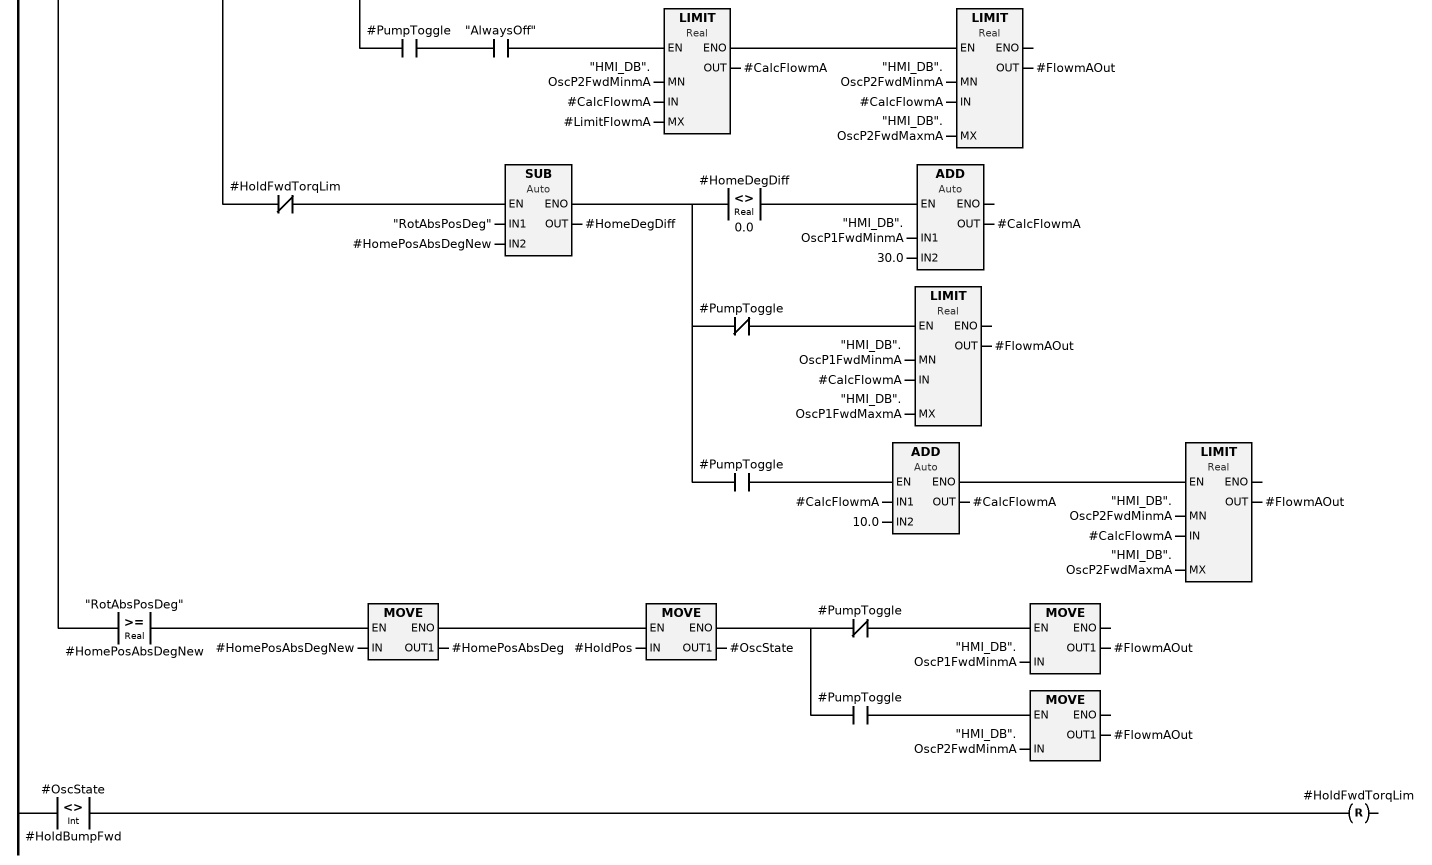
   RUNG wire#powerrail
      { S7_Templates := "SrcType := Int" } EQ_Contact(in1 := #OscState, in2 := #HoldBumpFwd)
      wire#w1
      Contact( #Oscillating )
      wire#w2
      P_Trig( #BumpFwdTrig )
      Move(in := "RotAbsPosDeg", out1 => #StartDeg)
      wire#w3
      I_Contact( #PumpToggle )
      Move(in := "HMI_DB".OscP1FwdMinmA, out1 => #CalcFlowmA)
   END_RUNG
   RUNG wire#w1
      Contact( #Holding )
   END_RUNG wire#w2
   RUNG wire#w3
      Contact( #PumpToggle )
      Move(in := "HMI_DB".OscP2FwdMinmA, out1 => #CalcFlowmA)
   END_RUNG
   RUNG wire#w2
      R_Coil( #FlowRev )
   END_RUNG
   RUNG wire#w2
      R_Coil( "HMI_DB".OscBumpFwd )
   END_RUNG
   RUNG wire#w2
      { S7_Templates := "SrcType := Real" } LT_Contact(in1 := "RotAbsPosDeg", in2 := #HomePosAbsDegNew)
      wire#w4
      { S7_Templates := "SrcType := Real" } GE_Contact(in1 := "ActTorqFtLbsFilt", in2 := "HMI_DB".OscTorqFwdLowLimFtlbs)
      { S7_Templates := "time_type := Time" } #HoldFWDTorqLim_TON.TON(pt := "Settings".OscTorqLimTime, et =>)
      S_Coil( #HoldFwdTorqLim )
   END_RUNG
   RUNG wire#w4
      { S7_Templates := "SrcType := Real" } GE_Contact(in1 := "ActTorqFtLbsFilt", in2 := "HMI_DB".OscTorqFwdHighLimFtLbs)
      S_Coil( #HoldFwdTorqLim )
   END_RUNG
   RUNG wire#w4
      Contact( #HoldFwdTorqLim )
      P_Trig( #HoldFwdTorqLimTrig )
      Move(in := #CalcFlowmA, out1 => #LimitFlowmA)
   END_RUNG
   RUNG wire#w4
      { S7_Templates := "SrcType := Real" } LT_Contact(in1 := "ActTorqFtLbsFilt", in2 := "HMI_DB".OscTorqFwdLowLimFtlbs)
      { S7_Templates := "SrcType := Real" } LT_Contact(in1 := #CalcFlowmA, in2 := #LimitFlowmA)
      R_Coil( #HoldFwdTorqLim )
   END_RUNG
   RUNG wire#w4
      Contact( #HoldFwdTorqLim )
      wire#w5
      { S7_Templates := "SrcType := Real" } GE_Contact(in1 := "ActTorqFtLbsFilt", in2 := "HMI_DB".OscTorqFwdHighLimFtLbs)
      Contact( "AlwaysOff" )
      #HoldFwdTorqLim_SlewDec(SlewRate := "HMI_DB".OscSlewFallSlow, RealValue := #LimitFlowmA)
   END_RUNG
   RUNG wire#w5
      { S7_Templates := "SrcType := Real" } LT_Contact(in1 := "ActTorqFtLbsFilt", in2 := "HMI_DB".OscTorqFwdLowLimFtlbs)
      Contact( "AlwaysOff" )
      #HoldFwdTorqLim_SlewInc(SlewRate := "HMI_DB".OscSlewRiseSlow, RealValue := #LimitFlowmA)
   END_RUNG
   RUNG wire#w5
      I_Contact( #PumpToggle )
      Contact( "AlwaysOff" )
      { S7_Templates := "value_type := Real" } Limit(mn := "HMI_DB".OscP1FwdMinmA, in := #CalcFlowmA, mx := #LimitFlowmA, out => #CalcFlowmA)
      { S7_Templates := "value_type := Real" } Limit(mn := "HMI_DB".OscP1FwdMinmA, in := #CalcFlowmA, mx := "HMI_DB".OscP1FwdMaxmA, out => #FlowmAOut)
   END_RUNG
   RUNG wire#w5
      Contact( #PumpToggle )
      Contact( "AlwaysOff" )
      { S7_Templates := "value_type := Real" } Limit(mn := "HMI_DB".OscP2FwdMinmA, in := #CalcFlowmA, mx := #LimitFlowmA, out => #CalcFlowmA)
      { S7_Templates := "value_type := Real" } Limit(mn := "HMI_DB".OscP2FwdMinmA, in := #CalcFlowmA, mx := "HMI_DB".OscP2FwdMaxmA, out => #FlowmAOut)
   END_RUNG
   RUNG wire#w4
      I_Contact( #HoldFwdTorqLim )
      Sub(in1 := "RotAbsPosDeg", in2 := #HomePosAbsDegNew, out => #HomeDegDiff)
      wire#w6
      { S7_Templates := "SrcType := Real" } NE_Contact(in1 := #HomeDegDiff, in2 := 0.0)
      Add(in1 := "HMI_DB".OscP1FwdMinmA, in2 := 30.0, out => #CalcFlowmA)
   END_RUNG
   RUNG wire#w6
      I_Contact( #PumpToggle )
      { S7_Templates := "value_type := Real" } Limit(mn := "HMI_DB".OscP1FwdMinmA, in := #CalcFlowmA, mx := "HMI_DB".OscP1FwdMaxmA, out => #FlowmAOut)
   END_RUNG
   RUNG wire#w6
      Contact( #PumpToggle )
      Add(in1 := #CalcFlowmA, in2 := 10.0, out => #CalcFlowmA)
      { S7_Templates := "value_type := Real" } Limit(mn := "HMI_DB".OscP2FwdMinmA, in := #CalcFlowmA, mx := "HMI_DB".OscP2FwdMaxmA, out => #FlowmAOut)
   END_RUNG
   RUNG wire#w2
      { S7_Templates := "SrcType := Real" } GE_Contact(in1 := "RotAbsPosDeg", in2 := #HomePosAbsDegNew)
      Move(in := #HomePosAbsDegNew, out1 => #HomePosAbsDeg)
      Move(in := #HoldPos, out1 => #OscState)
      wire#w7
      I_Contact( #PumpToggle )
      Move(in := "HMI_DB".OscP1FwdMinmA, out1 => #FlowmAOut)
   END_RUNG
   RUNG wire#w7
      Contact( #PumpToggle )
      Move(in := "HMI_DB".OscP2FwdMinmA, out1 => #FlowmAOut)
   END_RUNG
   RUNG wire#powerrail
      { S7_Templates := "SrcType := Int" } NE_Contact(in1 := #OscState, in2 := #HoldBumpFwd)
      R_Coil( #HoldFwdTorqLim )
   END_RUNG
   // the same network as SCL:
   #_w1 := (#OscState = #HoldBumpFwd) AND (#Oscillating OR #Holding);
   #_w2 := #_w1 AND NOT #BumpFwdTrig;   // rising edge
   #BumpFwdTrig := #_w1;
   IF #_w2 THEN #StartDeg := "RotAbsPosDeg"; END_IF;
   IF #_w2 AND NOT #PumpToggle THEN #CalcFlowmA := "HMI_DB".OscP1FwdMinmA; END_IF;
   IF #_w2 AND #PumpToggle THEN #CalcFlowmA := "HMI_DB".OscP2FwdMinmA; END_IF;
   IF #_w1 THEN
       #FlowRev := FALSE;
       "HMI_DB".OscBumpFwd := FALSE;
   END_IF;
   #_w3 := #_w1 AND ("RotAbsPosDeg" < #HomePosAbsDegNew);
   #HoldFWDTorqLim_TON(IN := #_w3 AND ("ActTorqFtLbsFilt" >= "HMI_DB".OscTorqFwdLowLimFtlbs),   // TON
                       PT := "Settings".OscTorqLimTime);
   IF #HoldFWDTorqLim_TON.Q THEN #HoldFwdTorqLim := TRUE; END_IF;
   IF #_w3 AND ("ActTorqFtLbsFilt" >= "HMI_DB".OscTorqFwdHighLimFtLbs) THEN #HoldFwdTorqLim := TRUE; END_IF;
   #_w4 := #_w3 AND #HoldFwdTorqLim;
   #_w5 := #_w4 AND NOT #HoldFwdTorqLimTrig;   // rising edge
   #HoldFwdTorqLimTrig := #_w4;
   IF #_w5 THEN #LimitFlowmA := #CalcFlowmA; END_IF;
   IF #_w3 AND ("ActTorqFtLbsFilt" < "HMI_DB".OscTorqFwdLowLimFtlbs) AND (#CalcFlowmA < #LimitFlowmA) THEN
       #HoldFwdTorqLim := FALSE;
   END_IF;
   #_w6 := #_w3 AND #HoldFwdTorqLim;
   IF #_w6 AND ("ActTorqFtLbsFilt" >= "HMI_DB".OscTorqFwdHighLimFtLbs) AND "AlwaysOff" THEN
       #HoldFwdTorqLim_SlewDec(SlewRate := "HMI_DB".OscSlewFallSlow, RealValue := #LimitFlowmA);   // "SlewDec"
   END_IF;
   IF #_w6 AND ("ActTorqFtLbsFilt" < "HMI_DB".OscTorqFwdLowLimFtlbs) AND "AlwaysOff" THEN
       #HoldFwdTorqLim_SlewInc(SlewRate := "HMI_DB".OscSlewRiseSlow, RealValue := #LimitFlowmA);   // "SlewInc"
   END_IF;
   IF #_w6 AND NOT #PumpToggle AND "AlwaysOff" THEN
       #CalcFlowmA := LIMIT(MN := "HMI_DB".OscP1FwdMinmA, IN := #CalcFlowmA, MX := #LimitFlowmA);
       #FlowmAOut := LIMIT(MN := "HMI_DB".OscP1FwdMinmA, IN := #CalcFlowmA, MX := "HMI_DB".OscP1FwdMaxmA);
   END_IF;
   IF #_w6 AND #PumpToggle AND "AlwaysOff" THEN
       #CalcFlowmA := LIMIT(MN := "HMI_DB".OscP2FwdMinmA, IN := #CalcFlowmA, MX := #LimitFlowmA);
       #FlowmAOut := LIMIT(MN := "HMI_DB".OscP2FwdMinmA, IN := #CalcFlowmA, MX := "HMI_DB".OscP2FwdMaxmA);
   END_IF;
   #_w7 := #_w3 AND NOT #HoldFwdTorqLim;
   IF #_w7 THEN #HomeDegDiff := "RotAbsPosDeg" - #HomePosAbsDegNew; END_IF;
   IF #_w7 AND (#HomeDegDiff <> 0.0) THEN #CalcFlowmA := "HMI_DB".OscP1FwdMinmA + 30.0; END_IF;
   IF #_w7 AND NOT #PumpToggle THEN
       #FlowmAOut := LIMIT(MN := "HMI_DB".OscP1FwdMinmA, IN := #CalcFlowmA, MX := "HMI_DB".OscP1FwdMaxmA);
   END_IF;
   IF #_w7 AND #PumpToggle THEN
       #CalcFlowmA := #CalcFlowmA + 10.0;
       #FlowmAOut := LIMIT(MN := "HMI_DB".OscP2FwdMinmA, IN := #CalcFlowmA, MX := "HMI_DB".OscP2FwdMaxmA);
   END_IF;
   #_w8 := #_w1 AND ("RotAbsPosDeg" >= #HomePosAbsDegNew);
   IF #_w8 THEN
       #HomePosAbsDeg := #HomePosAbsDegNew;
       #OscState := #HoldPos;
   END_IF;
   IF #_w8 AND NOT #PumpToggle THEN #FlowmAOut := "HMI_DB".OscP1FwdMinmA; END_IF;
   IF #_w8 AND #PumpToggle THEN #FlowmAOut := "HMI_DB".OscP2FwdMinmA; END_IF;
   IF #OscState <> #HoldBumpFwd THEN #HoldFwdTorqLim := FALSE; END_IF;
END_REGION

REGION Network 11: Hold Bump Reactive - State 104
   // Allow the quill to reactively move to the new position. 
   // Flow Rev enabled to Min until at Home position. If position below start position, min too high and moving wrong direction. Not reacting.  
   // At or above new home position, hold position
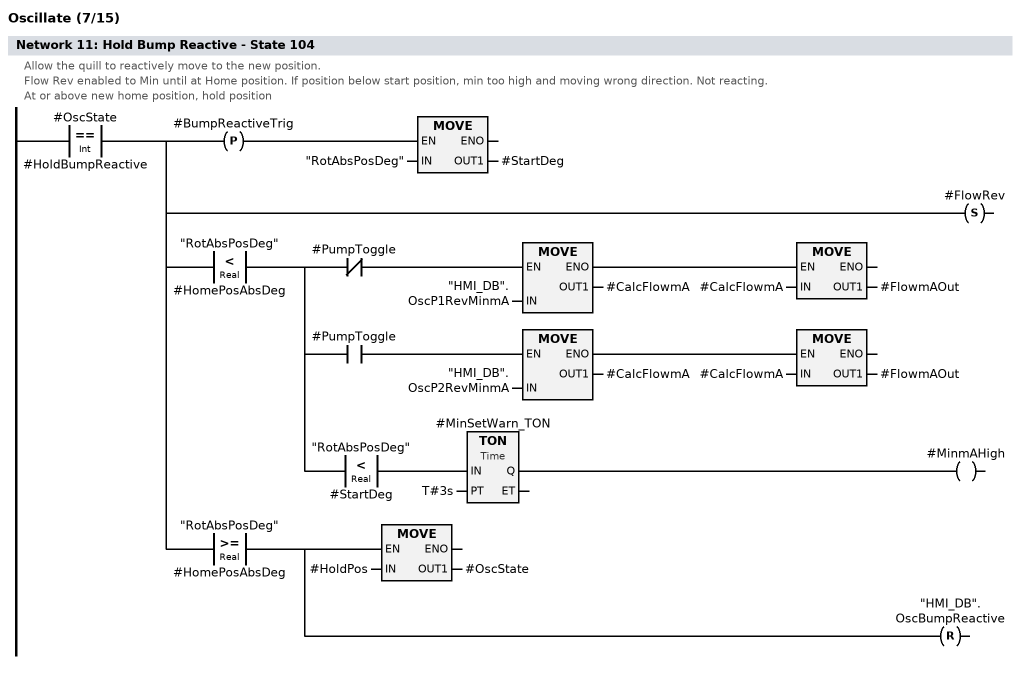
   RUNG wire#powerrail
      { S7_Templates := "SrcType := Int" } EQ_Contact(in1 := #OscState, in2 := #HoldBumpReactive)
      wire#w1
      P_Trig( #BumpReactiveTrig )
      Move(in := "RotAbsPosDeg", out1 => #StartDeg)
   END_RUNG
   RUNG wire#w1
      S_Coil( #FlowRev )
   END_RUNG
   RUNG wire#w1
      { S7_Templates := "SrcType := Real" } LT_Contact(in1 := "RotAbsPosDeg", in2 := #HomePosAbsDeg)
      wire#w2
      I_Contact( #PumpToggle )
      Move(in := "HMI_DB".OscP1RevMinmA, out1 => #CalcFlowmA)
      Move(in := #CalcFlowmA, out1 => #FlowmAOut)
   END_RUNG
   RUNG wire#w2
      Contact( #PumpToggle )
      Move(in := "HMI_DB".OscP2RevMinmA, out1 => #CalcFlowmA)
      Move(in := #CalcFlowmA, out1 => #FlowmAOut)
   END_RUNG
   RUNG wire#w2
      { S7_Templates := "SrcType := Real" } LT_Contact(in1 := "RotAbsPosDeg", in2 := #StartDeg)
      { S7_Templates := "time_type := Time" } #MinSetWarn_TON.TON(pt := T#3s, et =>)
      Coil( #MinmAHigh )
   END_RUNG
   RUNG wire#w1
      { S7_Templates := "SrcType := Real" } GE_Contact(in1 := "RotAbsPosDeg", in2 := #HomePosAbsDeg)
      wire#w3
      Move(in := #HoldPos, out1 => #OscState)
   END_RUNG
   RUNG wire#w3
      R_Coil( "HMI_DB".OscBumpReactive )
   END_RUNG
   // the same network as SCL:
   #_w1 := #OscState = #HoldBumpReactive;
   #_w2 := #_w1 AND NOT #BumpReactiveTrig;   // rising edge
   #BumpReactiveTrig := #_w1;
   IF #_w2 THEN #StartDeg := "RotAbsPosDeg"; END_IF;
   IF #_w1 THEN #FlowRev := TRUE; END_IF;
   #_w3 := #_w1 AND ("RotAbsPosDeg" < #HomePosAbsDeg);
   IF #_w3 AND NOT #PumpToggle THEN
       #CalcFlowmA := "HMI_DB".OscP1RevMinmA;
       #FlowmAOut := #CalcFlowmA;
   END_IF;
   IF #_w3 AND #PumpToggle THEN
       #CalcFlowmA := "HMI_DB".OscP2RevMinmA;
       #FlowmAOut := #CalcFlowmA;
   END_IF;
   #MinSetWarn_TON(IN := #_w3 AND ("RotAbsPosDeg" < #StartDeg), PT := T#3s);   // TON
   #MinmAHigh := #MinSetWarn_TON.Q;
   IF #_w1 AND ("RotAbsPosDeg" >= #HomePosAbsDeg) THEN
       #OscState := #HoldPos;
       "HMI_DB".OscBumpReactive := FALSE;
   END_IF;
END_REGION

REGION Network 12: Hold Bump Rev - State 103
   // Move quill to new position in the Rev direction. 
   // Start at Hold mA and Ramp up until speed reach. 
   // If Approaching Torq Limit, limit output flow. 
   // At or above new home position, output hold value and hold position
   // Note: Dummy Move On Maintain speed there as visual only.
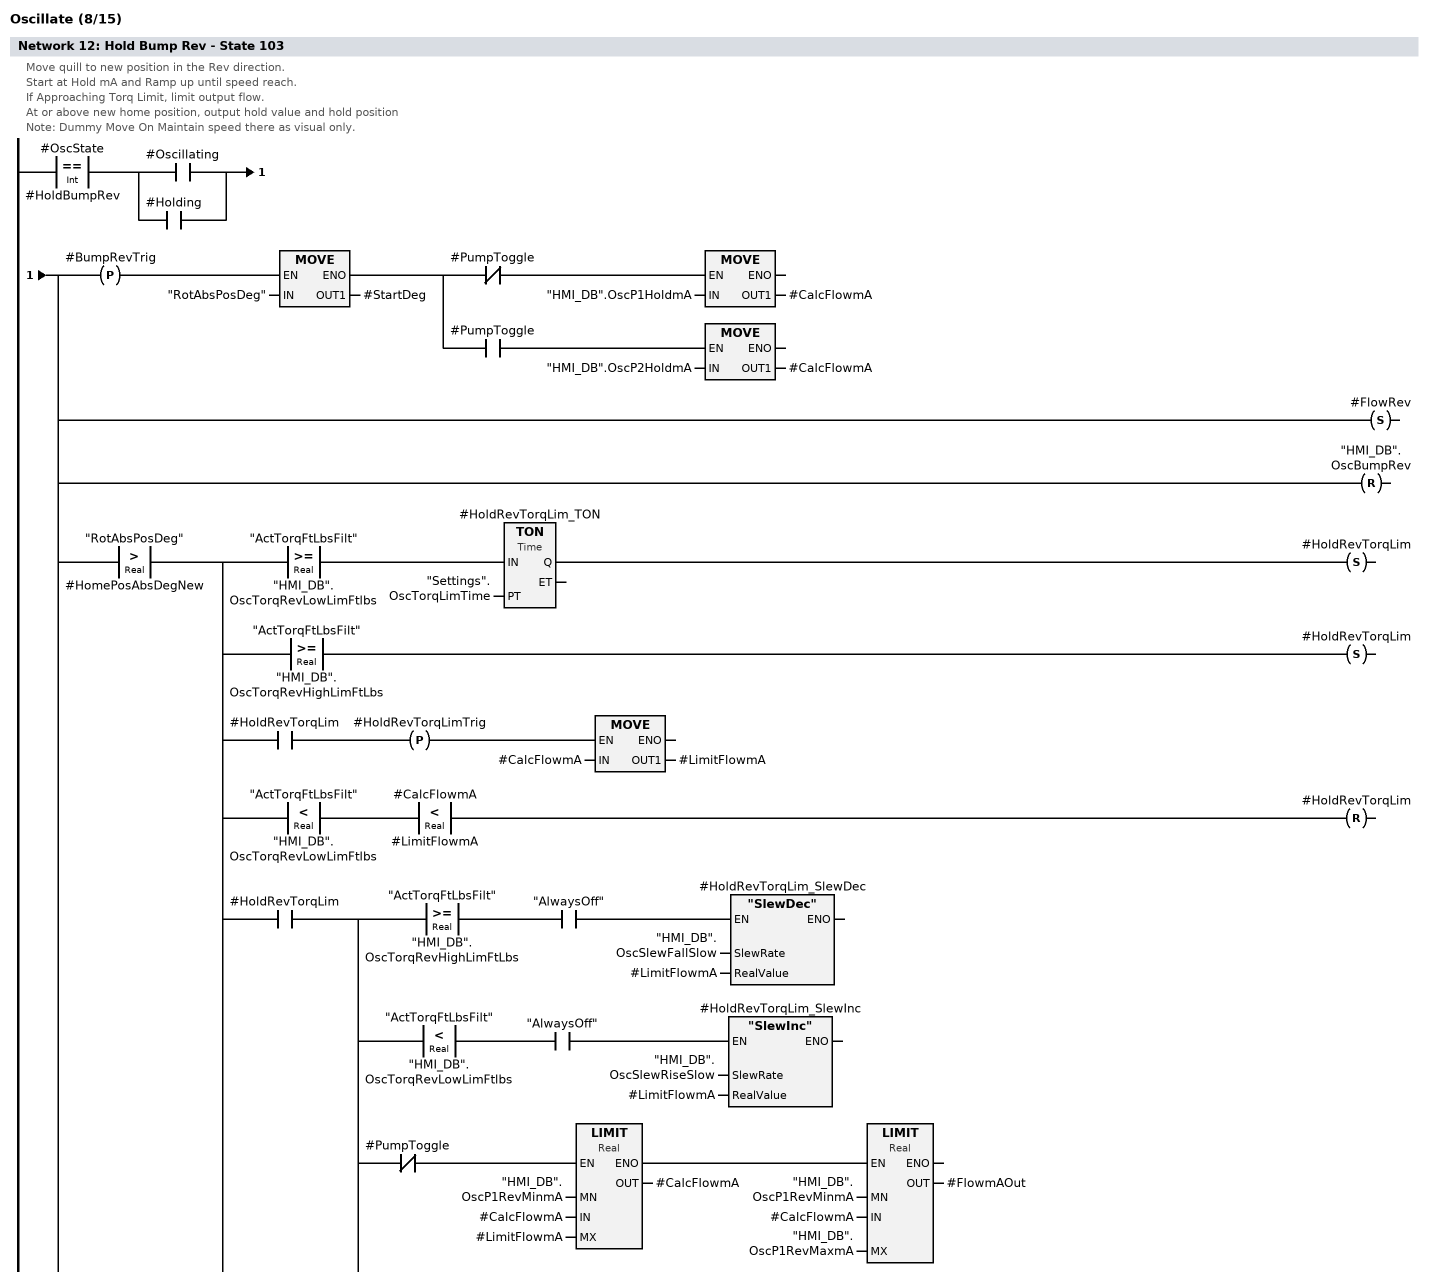
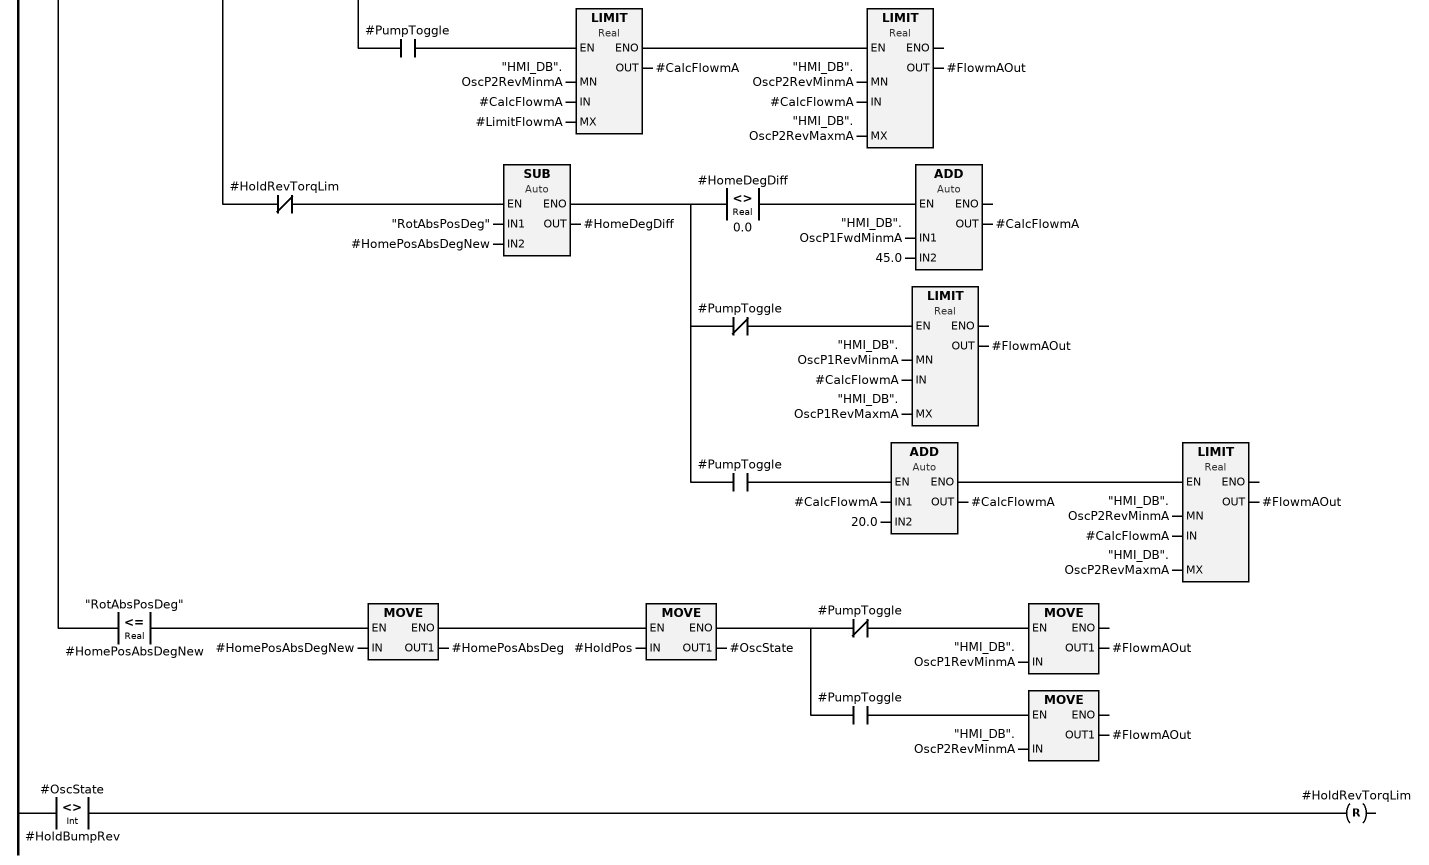
   RUNG wire#powerrail
      { S7_Templates := "SrcType := Int" } EQ_Contact(in1 := #OscState, in2 := #HoldBumpRev)
      wire#w1
      Contact( #Oscillating )
      wire#w2
      P_Trig( #BumpRevTrig )
      Move(in := "RotAbsPosDeg", out1 => #StartDeg)
      wire#w3
      I_Contact( #PumpToggle )
      Move(in := "HMI_DB".OscP1HoldmA, out1 => #CalcFlowmA)
   END_RUNG
   RUNG wire#w1
      Contact( #Holding )
   END_RUNG wire#w2
   RUNG wire#w3
      Contact( #PumpToggle )
      Move(in := "HMI_DB".OscP2HoldmA, out1 => #CalcFlowmA)
   END_RUNG
   RUNG wire#w2
      S_Coil( #FlowRev )
   END_RUNG
   RUNG wire#w2
      R_Coil( "HMI_DB".OscBumpRev )
   END_RUNG
   RUNG wire#w2
      { S7_Templates := "SrcType := Real" } GT_Contact(in1 := "RotAbsPosDeg", in2 := #HomePosAbsDegNew)
      wire#w4
      { S7_Templates := "SrcType := Real" } GE_Contact(in1 := "ActTorqFtLbsFilt", in2 := "HMI_DB".OscTorqRevLowLimFtlbs)
      { S7_Templates := "time_type := Time" } #HoldRevTorqLim_TON.TON(pt := "Settings".OscTorqLimTime, et =>)
      S_Coil( #HoldRevTorqLim )
   END_RUNG
   RUNG wire#w4
      { S7_Templates := "SrcType := Real" } GE_Contact(in1 := "ActTorqFtLbsFilt", in2 := "HMI_DB".OscTorqRevHighLimFtLbs)
      S_Coil( #HoldRevTorqLim )
   END_RUNG
   RUNG wire#w4
      Contact( #HoldRevTorqLim )
      P_Trig( #HoldRevTorqLimTrig )
      Move(in := #CalcFlowmA, out1 => #LimitFlowmA)
   END_RUNG
   RUNG wire#w4
      { S7_Templates := "SrcType := Real" } LT_Contact(in1 := "ActTorqFtLbsFilt", in2 := "HMI_DB".OscTorqRevLowLimFtlbs)
      { S7_Templates := "SrcType := Real" } LT_Contact(in1 := #CalcFlowmA, in2 := #LimitFlowmA)
      R_Coil( #HoldRevTorqLim )
   END_RUNG
   RUNG wire#w4
      Contact( #HoldRevTorqLim )
      wire#w5
      { S7_Templates := "SrcType := Real" } GE_Contact(in1 := "ActTorqFtLbsFilt", in2 := "HMI_DB".OscTorqRevHighLimFtLbs)
      Contact( "AlwaysOff" )
      #HoldRevTorqLim_SlewDec(SlewRate := "HMI_DB".OscSlewFallSlow, RealValue := #LimitFlowmA)
   END_RUNG
   RUNG wire#w5
      { S7_Templates := "SrcType := Real" } LT_Contact(in1 := "ActTorqFtLbsFilt", in2 := "HMI_DB".OscTorqRevLowLimFtlbs)
      Contact( "AlwaysOff" )
      #HoldRevTorqLim_SlewInc(SlewRate := "HMI_DB".OscSlewRiseSlow, RealValue := #LimitFlowmA)
   END_RUNG
   RUNG wire#w5
      I_Contact( #PumpToggle )
      { S7_Templates := "value_type := Real" } Limit(mn := "HMI_DB".OscP1RevMinmA, in := #CalcFlowmA, mx := #LimitFlowmA, out => #CalcFlowmA)
      { S7_Templates := "value_type := Real" } Limit(mn := "HMI_DB".OscP1RevMinmA, in := #CalcFlowmA, mx := "HMI_DB".OscP1RevMaxmA, out => #FlowmAOut)
   END_RUNG
   RUNG wire#w5
      Contact( #PumpToggle )
      { S7_Templates := "value_type := Real" } Limit(mn := "HMI_DB".OscP2RevMinmA, in := #CalcFlowmA, mx := #LimitFlowmA, out => #CalcFlowmA)
      { S7_Templates := "value_type := Real" } Limit(mn := "HMI_DB".OscP2RevMinmA, in := #CalcFlowmA, mx := "HMI_DB".OscP2RevMaxmA, out => #FlowmAOut)
   END_RUNG
   RUNG wire#w4
      I_Contact( #HoldRevTorqLim )
      Sub(in1 := "RotAbsPosDeg", in2 := #HomePosAbsDegNew, out => #HomeDegDiff)
      wire#w6
      { S7_Templates := "SrcType := Real" } NE_Contact(in1 := #HomeDegDiff, in2 := 0.0)
      Add(in1 := "HMI_DB".OscP1FwdMinmA, in2 := 45.0, out => #CalcFlowmA)
   END_RUNG
   RUNG wire#w6
      I_Contact( #PumpToggle )
      { S7_Templates := "value_type := Real" } Limit(mn := "HMI_DB".OscP1RevMinmA, in := #CalcFlowmA, mx := "HMI_DB".OscP1RevMaxmA, out => #FlowmAOut)
   END_RUNG
   RUNG wire#w6
      Contact( #PumpToggle )
      Add(in1 := #CalcFlowmA, in2 := 20.0, out => #CalcFlowmA)
      { S7_Templates := "value_type := Real" } Limit(mn := "HMI_DB".OscP2RevMinmA, in := #CalcFlowmA, mx := "HMI_DB".OscP2RevMaxmA, out => #FlowmAOut)
   END_RUNG
   RUNG wire#w2
      { S7_Templates := "SrcType := Real" } LE_Contact(in1 := "RotAbsPosDeg", in2 := #HomePosAbsDegNew)
      Move(in := #HomePosAbsDegNew, out1 => #HomePosAbsDeg)
      Move(in := #HoldPos, out1 => #OscState)
      wire#w7
      I_Contact( #PumpToggle )
      Move(in := "HMI_DB".OscP1RevMinmA, out1 => #FlowmAOut)
   END_RUNG
   RUNG wire#w7
      Contact( #PumpToggle )
      Move(in := "HMI_DB".OscP2RevMinmA, out1 => #FlowmAOut)
   END_RUNG
   RUNG wire#powerrail
      { S7_Templates := "SrcType := Int" } NE_Contact(in1 := #OscState, in2 := #HoldBumpRev)
      R_Coil( #HoldRevTorqLim )
   END_RUNG
   // the same network as SCL:
   #_w1 := (#OscState = #HoldBumpRev) AND (#Oscillating OR #Holding);
   #_w2 := #_w1 AND NOT #BumpRevTrig;   // rising edge
   #BumpRevTrig := #_w1;
   IF #_w2 THEN #StartDeg := "RotAbsPosDeg"; END_IF;
   IF #_w2 AND NOT #PumpToggle THEN #CalcFlowmA := "HMI_DB".OscP1HoldmA; END_IF;
   IF #_w2 AND #PumpToggle THEN #CalcFlowmA := "HMI_DB".OscP2HoldmA; END_IF;
   IF #_w1 THEN
       #FlowRev := TRUE;
       "HMI_DB".OscBumpRev := FALSE;
   END_IF;
   #_w3 := #_w1 AND ("RotAbsPosDeg" > #HomePosAbsDegNew);
   #HoldRevTorqLim_TON(IN := #_w3 AND ("ActTorqFtLbsFilt" >= "HMI_DB".OscTorqRevLowLimFtlbs),   // TON
                       PT := "Settings".OscTorqLimTime);
   IF #HoldRevTorqLim_TON.Q THEN #HoldRevTorqLim := TRUE; END_IF;
   IF #_w3 AND ("ActTorqFtLbsFilt" >= "HMI_DB".OscTorqRevHighLimFtLbs) THEN #HoldRevTorqLim := TRUE; END_IF;
   #_w4 := #_w3 AND #HoldRevTorqLim;
   #_w5 := #_w4 AND NOT #HoldRevTorqLimTrig;   // rising edge
   #HoldRevTorqLimTrig := #_w4;
   IF #_w5 THEN #LimitFlowmA := #CalcFlowmA; END_IF;
   IF #_w3 AND ("ActTorqFtLbsFilt" < "HMI_DB".OscTorqRevLowLimFtlbs) AND (#CalcFlowmA < #LimitFlowmA) THEN
       #HoldRevTorqLim := FALSE;
   END_IF;
   #_w6 := #_w3 AND #HoldRevTorqLim;
   IF #_w6 AND ("ActTorqFtLbsFilt" >= "HMI_DB".OscTorqRevHighLimFtLbs) AND "AlwaysOff" THEN
       #HoldRevTorqLim_SlewDec(SlewRate := "HMI_DB".OscSlewFallSlow, RealValue := #LimitFlowmA);   // "SlewDec"
   END_IF;
   IF #_w6 AND ("ActTorqFtLbsFilt" < "HMI_DB".OscTorqRevLowLimFtlbs) AND "AlwaysOff" THEN
       #HoldRevTorqLim_SlewInc(SlewRate := "HMI_DB".OscSlewRiseSlow, RealValue := #LimitFlowmA);   // "SlewInc"
   END_IF;
   IF #_w6 AND NOT #PumpToggle THEN
       #CalcFlowmA := LIMIT(MN := "HMI_DB".OscP1RevMinmA, IN := #CalcFlowmA, MX := #LimitFlowmA);
       #FlowmAOut := LIMIT(MN := "HMI_DB".OscP1RevMinmA, IN := #CalcFlowmA, MX := "HMI_DB".OscP1RevMaxmA);
   END_IF;
   IF #_w6 AND #PumpToggle THEN
       #CalcFlowmA := LIMIT(MN := "HMI_DB".OscP2RevMinmA, IN := #CalcFlowmA, MX := #LimitFlowmA);
       #FlowmAOut := LIMIT(MN := "HMI_DB".OscP2RevMinmA, IN := #CalcFlowmA, MX := "HMI_DB".OscP2RevMaxmA);
   END_IF;
   #_w7 := #_w3 AND NOT #HoldRevTorqLim;
   IF #_w7 THEN #HomeDegDiff := "RotAbsPosDeg" - #HomePosAbsDegNew; END_IF;
   IF #_w7 AND (#HomeDegDiff <> 0.0) THEN #CalcFlowmA := "HMI_DB".OscP1FwdMinmA + 45.0; END_IF;
   IF #_w7 AND NOT #PumpToggle THEN
       #FlowmAOut := LIMIT(MN := "HMI_DB".OscP1RevMinmA, IN := #CalcFlowmA, MX := "HMI_DB".OscP1RevMaxmA);
   END_IF;
   IF #_w7 AND #PumpToggle THEN
       #CalcFlowmA := #CalcFlowmA + 20.0;
       #FlowmAOut := LIMIT(MN := "HMI_DB".OscP2RevMinmA, IN := #CalcFlowmA, MX := "HMI_DB".OscP2RevMaxmA);
   END_IF;
   #_w8 := #_w1 AND ("RotAbsPosDeg" <= #HomePosAbsDegNew);
   IF #_w8 THEN
       #HomePosAbsDeg := #HomePosAbsDegNew;
       #OscState := #HoldPos;
   END_IF;
   IF #_w8 AND NOT #PumpToggle THEN #FlowmAOut := "HMI_DB".OscP1RevMinmA; END_IF;
   IF #_w8 AND #PumpToggle THEN #FlowmAOut := "HMI_DB".OscP2RevMinmA; END_IF;
   IF #OscState <> #HoldBumpRev THEN #HoldRevTorqLim := FALSE; END_IF;
END_REGION

REGION Network 13: Start Oscillate - State 200
   // Toggel Pump Use when starting. Store starting values and calculate target positions
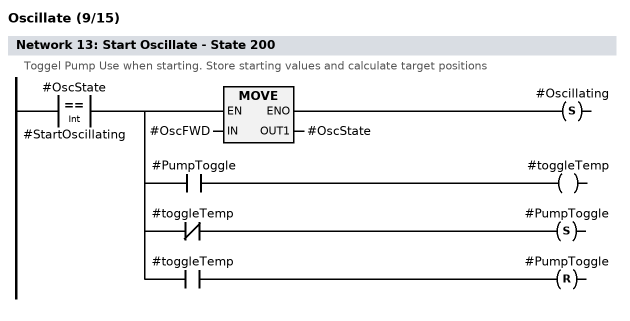
   RUNG wire#powerrail
      { S7_Templates := "SrcType := Int" } EQ_Contact(in1 := #OscState, in2 := #StartOscillating)
      wire#w1
      Move(in := #OscFWD, out1 => #OscState)
      S_Coil( #Oscillating )
   END_RUNG
   RUNG wire#w1
      Contact( #PumpToggle )
      Coil( #toggleTemp )
   END_RUNG
   RUNG wire#w1
      I_Contact( #toggleTemp )
      S_Coil( #PumpToggle )
   END_RUNG
   RUNG wire#w1
      Contact( #toggleTemp )
      R_Coil( #PumpToggle )
   END_RUNG
   // the same network as SCL:
   #_w1 := #OscState = #StartOscillating;
   IF #_w1 THEN
       #OscState := #OscFWD;
       #Oscillating := TRUE;
   END_IF;
   #toggleTemp := #_w1 AND #PumpToggle;
   IF #_w1 AND NOT #toggleTemp THEN #PumpToggle := TRUE; END_IF;
   IF #_w1 AND #toggleTemp THEN #PumpToggle := FALSE; END_IF;
END_REGION

REGION Network 14: Osc Fwd - State 201
   // Move quill to FWD end position in the FWD direction. 
   // Start at Min and Ramp up until speed reach. 
   // If Approaching Torq Limit, limit output flow. 
   // At or above end position, switch direction
   // Note: Dummy Move On Maintain speed there as visual only.
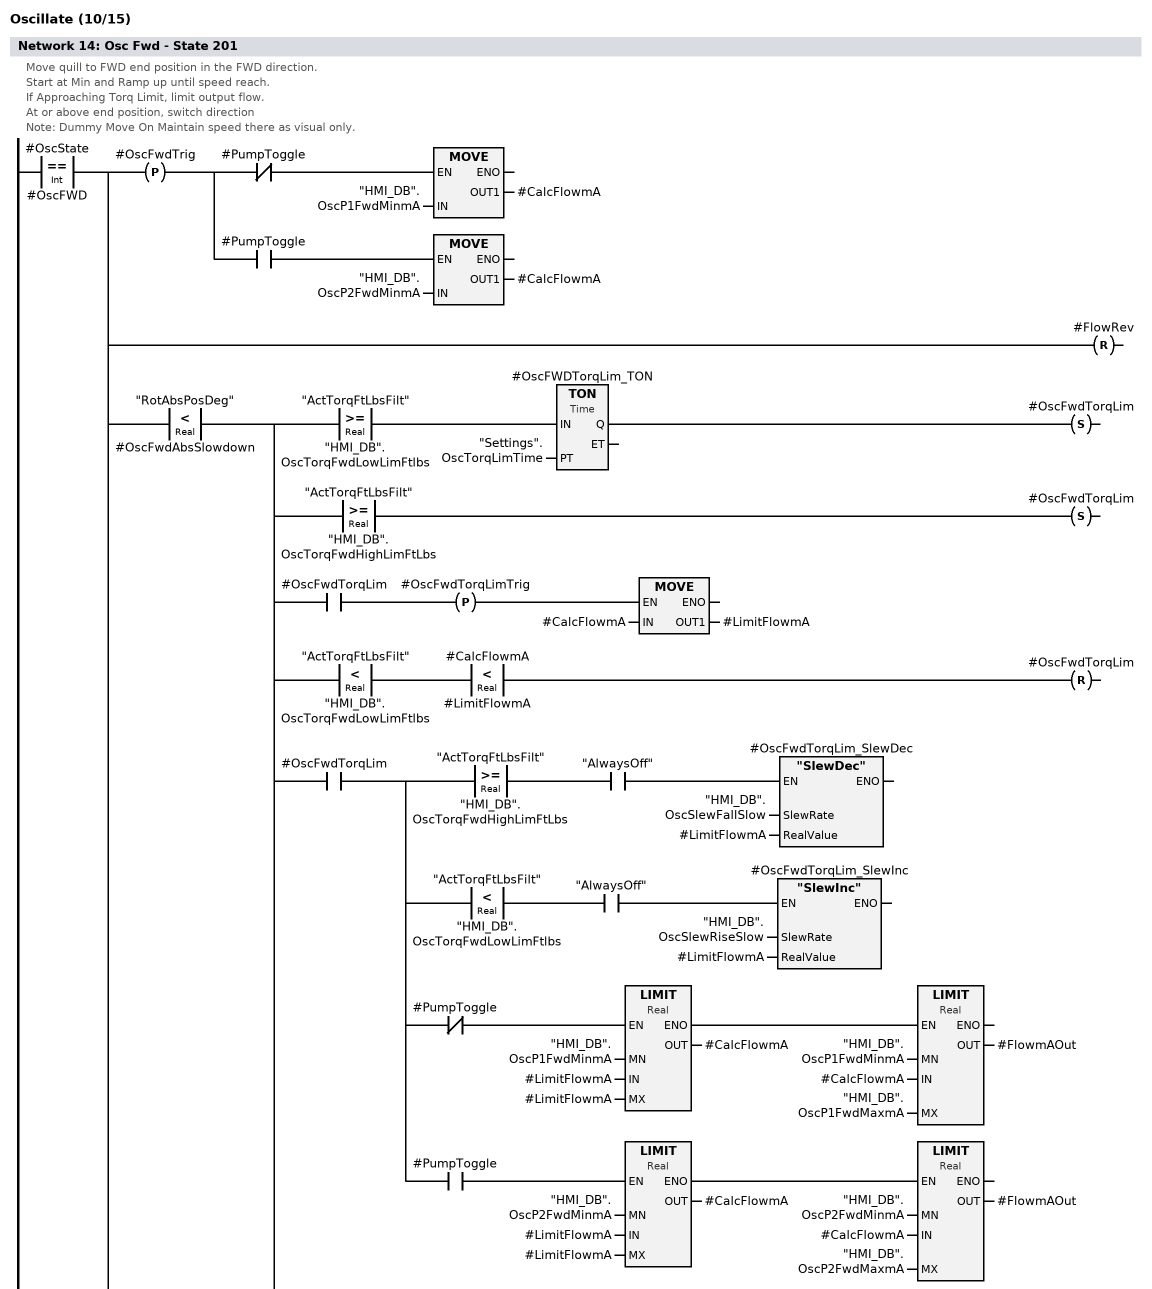
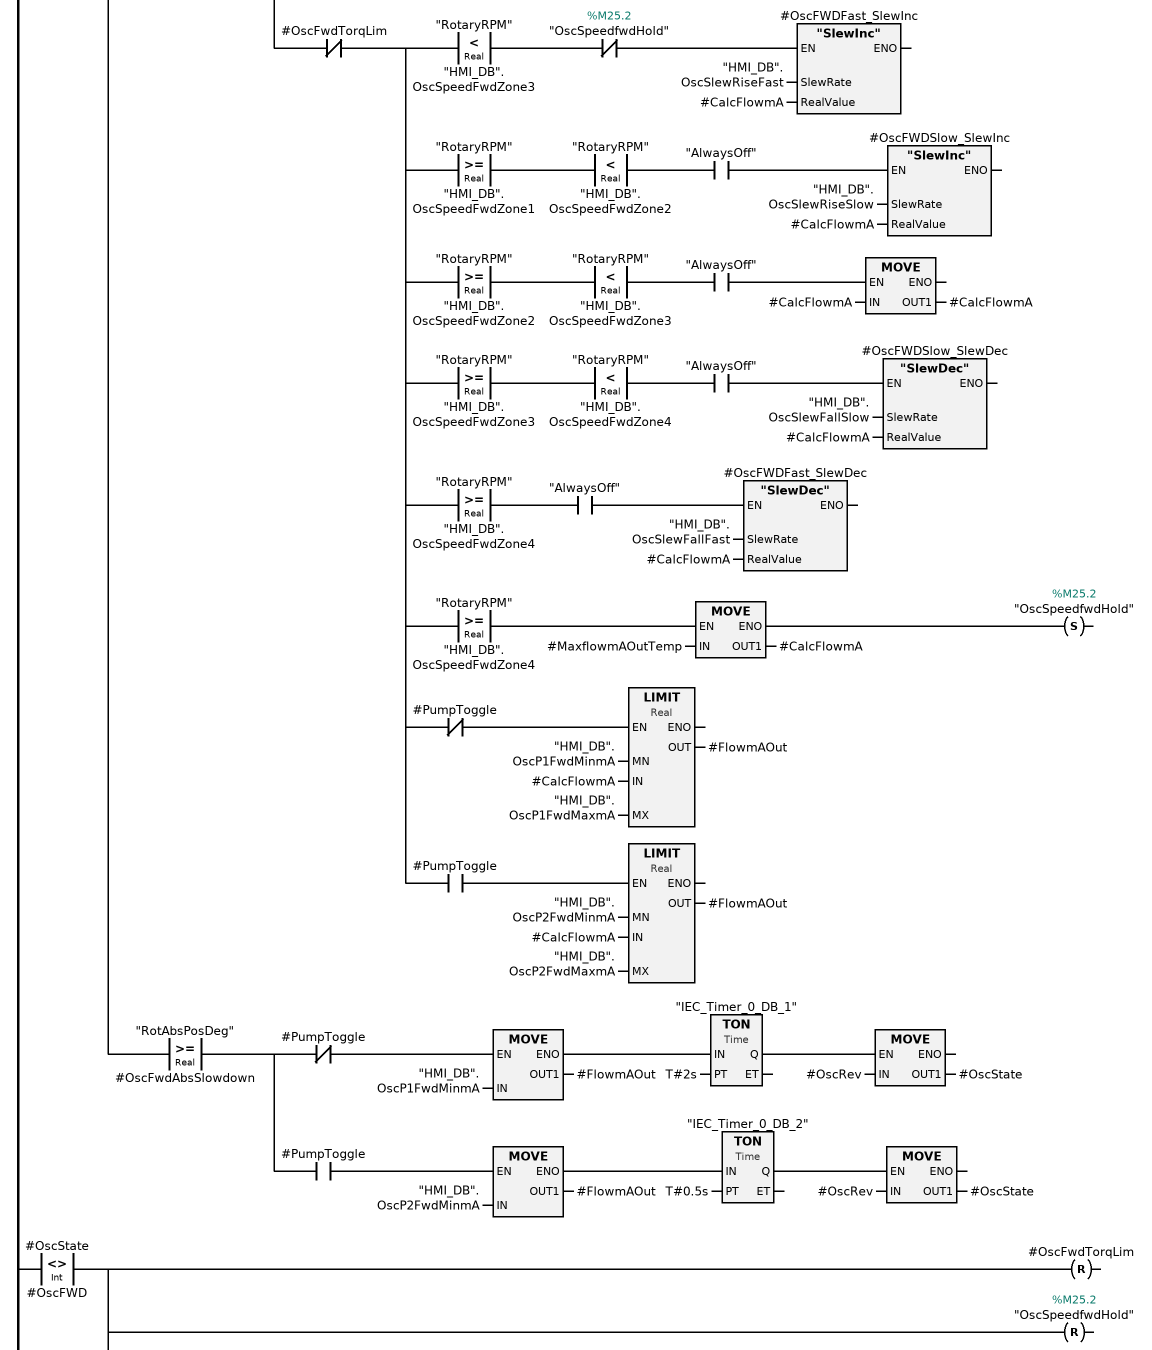
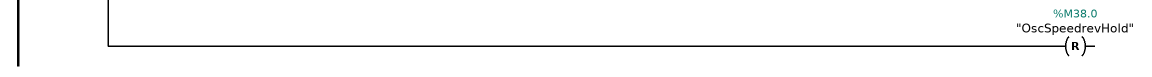
   RUNG wire#powerrail
      { S7_Templates := "SrcType := Int" } EQ_Contact(in1 := #OscState, in2 := #OscFWD)
      wire#w1
      P_Trig( #OscFwdTrig )
      wire#w2
      I_Contact( #PumpToggle )
      Move(in := "HMI_DB".OscP1FwdMinmA, out1 => #CalcFlowmA)
   END_RUNG
   RUNG wire#w2
      Contact( #PumpToggle )
      Move(in := "HMI_DB".OscP2FwdMinmA, out1 => #CalcFlowmA)
   END_RUNG
   RUNG wire#w1
      R_Coil( #FlowRev )
   END_RUNG
   RUNG wire#w1
      { S7_Templates := "SrcType := Real" } LT_Contact(in1 := "RotAbsPosDeg", in2 := #OscFwdAbsSlowdown)
      wire#w3
      { S7_Templates := "SrcType := Real" } GE_Contact(in1 := "ActTorqFtLbsFilt", in2 := "HMI_DB".OscTorqFwdLowLimFtlbs)
      { S7_Templates := "time_type := Time" } #OscFWDTorqLim_TON.TON(pt := "Settings".OscTorqLimTime, et =>)
      S_Coil( #OscFwdTorqLim )
   END_RUNG
   RUNG wire#w3
      { S7_Templates := "SrcType := Real" } GE_Contact(in1 := "ActTorqFtLbsFilt", in2 := "HMI_DB".OscTorqFwdHighLimFtLbs)
      S_Coil( #OscFwdTorqLim )
   END_RUNG
   RUNG wire#w3
      Contact( #OscFwdTorqLim )
      P_Trig( #OscFwdTorqLimTrig )
      Move(in := #CalcFlowmA, out1 => #LimitFlowmA)
   END_RUNG
   RUNG wire#w3
      { S7_Templates := "SrcType := Real" } LT_Contact(in1 := "ActTorqFtLbsFilt", in2 := "HMI_DB".OscTorqFwdLowLimFtlbs)
      { S7_Templates := "SrcType := Real" } LT_Contact(in1 := #CalcFlowmA, in2 := #LimitFlowmA)
      R_Coil( #OscFwdTorqLim )
   END_RUNG
   RUNG wire#w3
      Contact( #OscFwdTorqLim )
      wire#w4
      { S7_Templates := "SrcType := Real" } GE_Contact(in1 := "ActTorqFtLbsFilt", in2 := "HMI_DB".OscTorqFwdHighLimFtLbs)
      Contact( "AlwaysOff" )
      #OscFwdTorqLim_SlewDec(SlewRate := "HMI_DB".OscSlewFallSlow, RealValue := #LimitFlowmA)
   END_RUNG
   RUNG wire#w4
      { S7_Templates := "SrcType := Real" } LT_Contact(in1 := "ActTorqFtLbsFilt", in2 := "HMI_DB".OscTorqFwdLowLimFtlbs)
      Contact( "AlwaysOff" )
      #OscFwdTorqLim_SlewInc(SlewRate := "HMI_DB".OscSlewRiseSlow, RealValue := #LimitFlowmA)
   END_RUNG
   RUNG wire#w4
      I_Contact( #PumpToggle )
      { S7_Templates := "value_type := Real" } Limit(mn := "HMI_DB".OscP1FwdMinmA, in := #LimitFlowmA, mx := #LimitFlowmA, out => #CalcFlowmA)
      { S7_Templates := "value_type := Real" } Limit(mn := "HMI_DB".OscP1FwdMinmA, in := #CalcFlowmA, mx := "HMI_DB".OscP1FwdMaxmA, out => #FlowmAOut)
   END_RUNG
   RUNG wire#w4
      Contact( #PumpToggle )
      { S7_Templates := "value_type := Real" } Limit(mn := "HMI_DB".OscP2FwdMinmA, in := #LimitFlowmA, mx := #LimitFlowmA, out => #CalcFlowmA)
      { S7_Templates := "value_type := Real" } Limit(mn := "HMI_DB".OscP2FwdMinmA, in := #CalcFlowmA, mx := "HMI_DB".OscP2FwdMaxmA, out => #FlowmAOut)
   END_RUNG
   RUNG wire#w3
      I_Contact( #OscFwdTorqLim )
      wire#w5
      { S7_Templates := "SrcType := Real" } LT_Contact(in1 := "RotaryRPM", in2 := "HMI_DB".OscSpeedFwdZone3)
      I_Contact( "OscSpeedfwdHold" )
      #OscFWDFast_SlewInc(SlewRate := "HMI_DB".OscSlewRiseFast, RealValue := #CalcFlowmA)
   END_RUNG
   RUNG wire#w5
      { S7_Templates := "SrcType := Real" } GE_Contact(in1 := "RotaryRPM", in2 := "HMI_DB".OscSpeedFwdZone1)
      { S7_Templates := "SrcType := Real" } LT_Contact(in1 := "RotaryRPM", in2 := "HMI_DB".OscSpeedFwdZone2)
      Contact( "AlwaysOff" )
      #OscFWDSlow_SlewInc(SlewRate := "HMI_DB".OscSlewRiseSlow, RealValue := #CalcFlowmA)
   END_RUNG
   RUNG wire#w5
      { S7_Templates := "SrcType := Real" } GE_Contact(in1 := "RotaryRPM", in2 := "HMI_DB".OscSpeedFwdZone2)
      { S7_Templates := "SrcType := Real" } LT_Contact(in1 := "RotaryRPM", in2 := "HMI_DB".OscSpeedFwdZone3)
      Contact( "AlwaysOff" )
      Move(in := #CalcFlowmA, out1 => #CalcFlowmA)
   END_RUNG
   RUNG wire#w5
      { S7_Templates := "SrcType := Real" } GE_Contact(in1 := "RotaryRPM", in2 := "HMI_DB".OscSpeedFwdZone3)
      { S7_Templates := "SrcType := Real" } LT_Contact(in1 := "RotaryRPM", in2 := "HMI_DB".OscSpeedFwdZone4)
      Contact( "AlwaysOff" )
      #OscFWDSlow_SlewDec(SlewRate := "HMI_DB".OscSlewFallSlow, RealValue := #CalcFlowmA)
   END_RUNG
   RUNG wire#w5
      { S7_Templates := "SrcType := Real" } GE_Contact(in1 := "RotaryRPM", in2 := "HMI_DB".OscSpeedFwdZone4)
      Contact( "AlwaysOff" )
      #OscFWDFast_SlewDec(SlewRate := "HMI_DB".OscSlewFallFast, RealValue := #CalcFlowmA)
   END_RUNG
   RUNG wire#w5
      { S7_Templates := "SrcType := Real" } GE_Contact(in1 := "RotaryRPM", in2 := "HMI_DB".OscSpeedFwdZone4)
      Move(in := #MaxflowmAOutTemp, out1 => #CalcFlowmA)
      S_Coil( "OscSpeedfwdHold" )
   END_RUNG
   RUNG wire#w5
      I_Contact( #PumpToggle )
      { S7_Templates := "value_type := Real" } Limit(mn := "HMI_DB".OscP1FwdMinmA, in := #CalcFlowmA, mx := "HMI_DB".OscP1FwdMaxmA, out => #FlowmAOut)
   END_RUNG
   RUNG wire#w5
      Contact( #PumpToggle )
      { S7_Templates := "value_type := Real" } Limit(mn := "HMI_DB".OscP2FwdMinmA, in := #CalcFlowmA, mx := "HMI_DB".OscP2FwdMaxmA, out => #FlowmAOut)
   END_RUNG
   RUNG wire#w1
      { S7_Templates := "SrcType := Real" } GE_Contact(in1 := "RotAbsPosDeg", in2 := #OscFwdAbsSlowdown)
      wire#w6
      I_Contact( #PumpToggle )
      Move(in := "HMI_DB".OscP1FwdMinmA, out1 => #FlowmAOut)
      { S7_Templates := "time_type := Time" } "IEC_Timer_0_DB_1".TON(pt := T#2s, et =>)
      Move(in := #OscRev, out1 => #OscState)
   END_RUNG
   RUNG wire#w6
      Contact( #PumpToggle )
      Move(in := "HMI_DB".OscP2FwdMinmA, out1 => #FlowmAOut)
      { S7_Templates := "time_type := Time" } "IEC_Timer_0_DB_2".TON(pt := T#0.5s, et =>)
      Move(in := #OscRev, out1 => #OscState)
   END_RUNG
   RUNG wire#powerrail
      { S7_Templates := "SrcType := Int" } NE_Contact(in1 := #OscState, in2 := #OscFWD)
      wire#w7
      R_Coil( #OscFwdTorqLim )
   END_RUNG
   RUNG wire#w7
      R_Coil( "OscSpeedfwdHold" )
   END_RUNG
   RUNG wire#w7
      R_Coil( "OscSpeedrevHold" )
   END_RUNG
   // the same network as SCL:
   #_w1 := #OscState = #OscFWD;
   #_w2 := #_w1 AND NOT #OscFwdTrig;   // rising edge
   #OscFwdTrig := #_w1;
   IF #_w2 AND NOT #PumpToggle THEN #CalcFlowmA := "HMI_DB".OscP1FwdMinmA; END_IF;
   IF #_w2 AND #PumpToggle THEN #CalcFlowmA := "HMI_DB".OscP2FwdMinmA; END_IF;
   IF #_w1 THEN #FlowRev := FALSE; END_IF;
   #_w3 := #_w1 AND ("RotAbsPosDeg" < #OscFwdAbsSlowdown);
   #OscFWDTorqLim_TON(IN := #_w3 AND ("ActTorqFtLbsFilt" >= "HMI_DB".OscTorqFwdLowLimFtlbs),   // TON
                      PT := "Settings".OscTorqLimTime);
   IF #OscFWDTorqLim_TON.Q THEN #OscFwdTorqLim := TRUE; END_IF;
   IF #_w3 AND ("ActTorqFtLbsFilt" >= "HMI_DB".OscTorqFwdHighLimFtLbs) THEN #OscFwdTorqLim := TRUE; END_IF;
   #_w4 := #_w3 AND #OscFwdTorqLim;
   #_w5 := #_w4 AND NOT #OscFwdTorqLimTrig;   // rising edge
   #OscFwdTorqLimTrig := #_w4;
   IF #_w5 THEN #LimitFlowmA := #CalcFlowmA; END_IF;
   IF #_w3 AND ("ActTorqFtLbsFilt" < "HMI_DB".OscTorqFwdLowLimFtlbs) AND (#CalcFlowmA < #LimitFlowmA) THEN
       #OscFwdTorqLim := FALSE;
   END_IF;
   #_w6 := #_w3 AND #OscFwdTorqLim;
   IF #_w6 AND ("ActTorqFtLbsFilt" >= "HMI_DB".OscTorqFwdHighLimFtLbs) AND "AlwaysOff" THEN
       #OscFwdTorqLim_SlewDec(SlewRate := "HMI_DB".OscSlewFallSlow, RealValue := #LimitFlowmA);   // "SlewDec"
   END_IF;
   IF #_w6 AND ("ActTorqFtLbsFilt" < "HMI_DB".OscTorqFwdLowLimFtlbs) AND "AlwaysOff" THEN
       #OscFwdTorqLim_SlewInc(SlewRate := "HMI_DB".OscSlewRiseSlow, RealValue := #LimitFlowmA);   // "SlewInc"
   END_IF;
   IF #_w6 AND NOT #PumpToggle THEN
       #CalcFlowmA := LIMIT(MN := "HMI_DB".OscP1FwdMinmA, IN := #LimitFlowmA, MX := #LimitFlowmA);
       #FlowmAOut := LIMIT(MN := "HMI_DB".OscP1FwdMinmA, IN := #CalcFlowmA, MX := "HMI_DB".OscP1FwdMaxmA);
   END_IF;
   IF #_w6 AND #PumpToggle THEN
       #CalcFlowmA := LIMIT(MN := "HMI_DB".OscP2FwdMinmA, IN := #LimitFlowmA, MX := #LimitFlowmA);
       #FlowmAOut := LIMIT(MN := "HMI_DB".OscP2FwdMinmA, IN := #CalcFlowmA, MX := "HMI_DB".OscP2FwdMaxmA);
   END_IF;
   #_w7 := #_w3 AND NOT #OscFwdTorqLim;
   IF #_w7 AND ("RotaryRPM" < "HMI_DB".OscSpeedFwdZone3) AND NOT "OscSpeedfwdHold" THEN
       #OscFWDFast_SlewInc(SlewRate := "HMI_DB".OscSlewRiseFast, RealValue := #CalcFlowmA);   // "SlewInc"
   END_IF;
   IF #_w7 AND ("RotaryRPM" >= "HMI_DB".OscSpeedFwdZone1) AND ("RotaryRPM" < "HMI_DB".OscSpeedFwdZone2) AND "AlwaysOff" THEN
       #OscFWDSlow_SlewInc(SlewRate := "HMI_DB".OscSlewRiseSlow, RealValue := #CalcFlowmA);   // "SlewInc"
   END_IF;
   IF #_w7 AND ("RotaryRPM" >= "HMI_DB".OscSpeedFwdZone2) AND ("RotaryRPM" < "HMI_DB".OscSpeedFwdZone3) AND "AlwaysOff" THEN
       #CalcFlowmA := #CalcFlowmA;
   END_IF;
   IF #_w7 AND ("RotaryRPM" >= "HMI_DB".OscSpeedFwdZone3) AND ("RotaryRPM" < "HMI_DB".OscSpeedFwdZone4) AND "AlwaysOff" THEN
       #OscFWDSlow_SlewDec(SlewRate := "HMI_DB".OscSlewFallSlow, RealValue := #CalcFlowmA);   // "SlewDec"
   END_IF;
   IF #_w7 AND ("RotaryRPM" >= "HMI_DB".OscSpeedFwdZone4) AND "AlwaysOff" THEN
       #OscFWDFast_SlewDec(SlewRate := "HMI_DB".OscSlewFallFast, RealValue := #CalcFlowmA);   // "SlewDec"
   END_IF;
   IF #_w7 AND ("RotaryRPM" >= "HMI_DB".OscSpeedFwdZone4) THEN
       #CalcFlowmA := #MaxflowmAOutTemp;
       "OscSpeedfwdHold" := TRUE;
   END_IF;
   IF #_w7 AND NOT #PumpToggle THEN
       #FlowmAOut := LIMIT(MN := "HMI_DB".OscP1FwdMinmA, IN := #CalcFlowmA, MX := "HMI_DB".OscP1FwdMaxmA);
   END_IF;
   IF #_w7 AND #PumpToggle THEN
       #FlowmAOut := LIMIT(MN := "HMI_DB".OscP2FwdMinmA, IN := #CalcFlowmA, MX := "HMI_DB".OscP2FwdMaxmA);
   END_IF;
   #_w8 := #_w1 AND ("RotAbsPosDeg" >= #OscFwdAbsSlowdown);
   #_w9 := #_w8 AND NOT #PumpToggle;
   IF #_w9 THEN #FlowmAOut := "HMI_DB".OscP1FwdMinmA; END_IF;
   "IEC_Timer_0_DB_1".TON(IN := #_w9, PT := T#2s);
   IF "IEC_Timer_0_DB_1".Q THEN #OscState := #OscRev; END_IF;
   #_w10 := #_w8 AND #PumpToggle;
   IF #_w10 THEN #FlowmAOut := "HMI_DB".OscP2FwdMinmA; END_IF;
   "IEC_Timer_0_DB_2".TON(IN := #_w10, PT := T#0.5s);
   IF "IEC_Timer_0_DB_2".Q THEN #OscState := #OscRev; END_IF;
   IF #OscState <> #OscFWD THEN
       #OscFwdTorqLim := FALSE;
       "OscSpeedfwdHold" := FALSE;
       "OscSpeedrevHold" := FALSE;
   END_IF;
END_REGION

REGION Network 15: Osc Rev - State 202
   // Move quill to new position in the Rev direction. 
   // Start at Hold mA and Ramp up until speed reach. 
   // If Approaching Torq Limit, limit output flow. 
   // At or above new home position, output hold value and hold position
   // Note: Dummy Move On Maintain speed there as visual only.
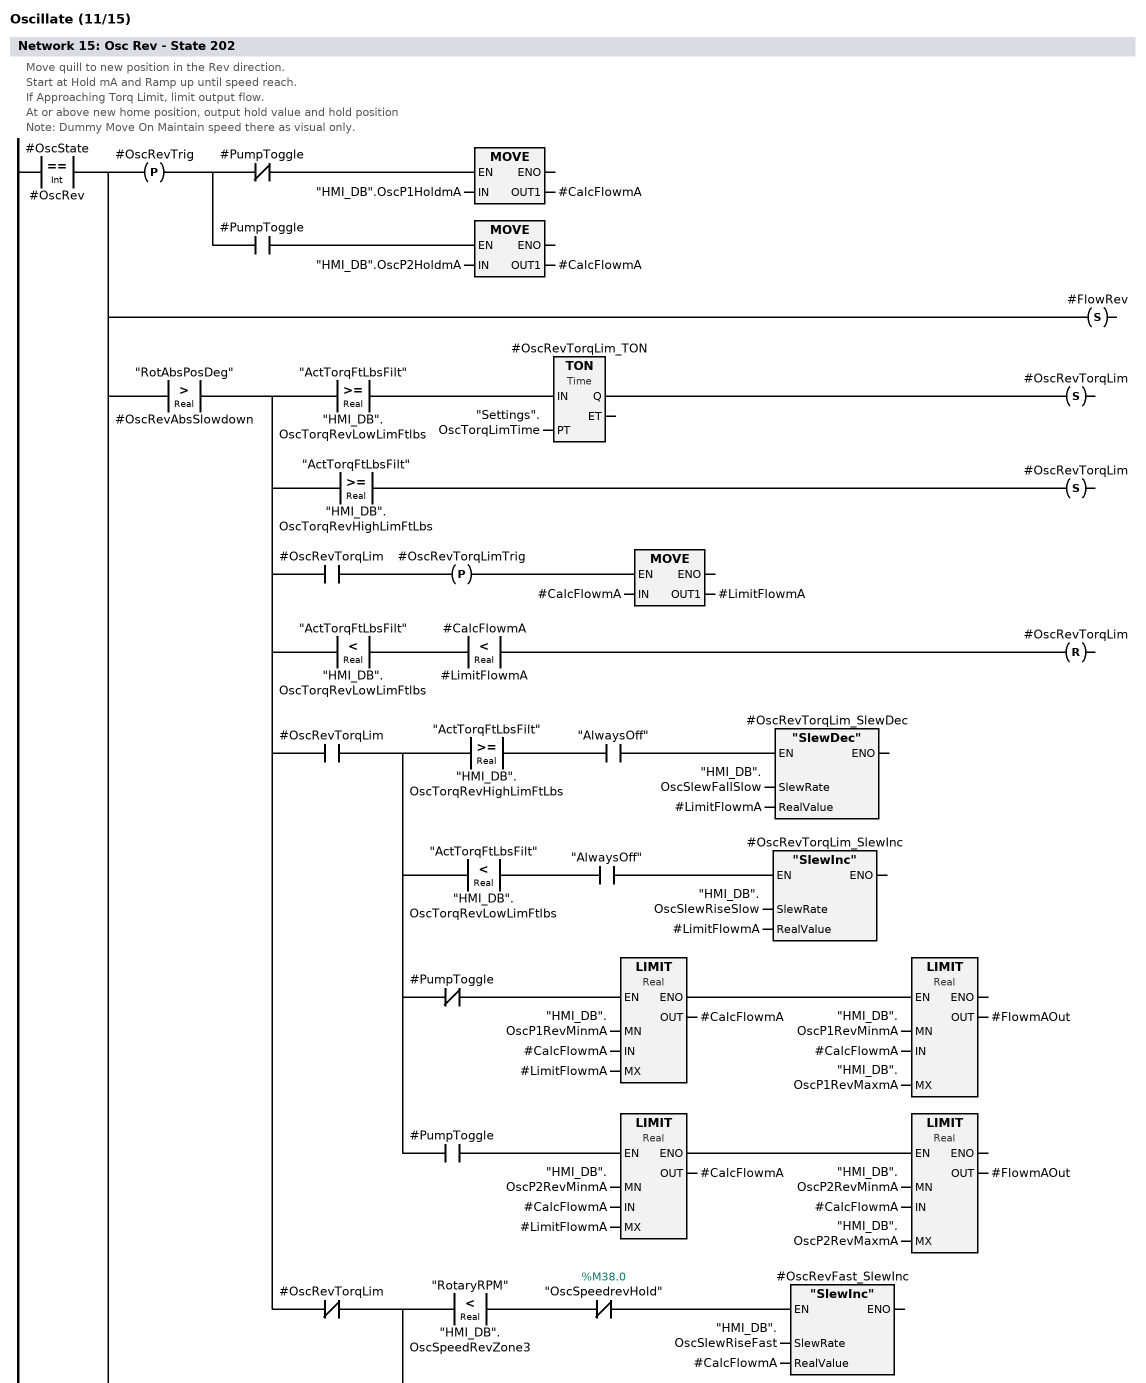
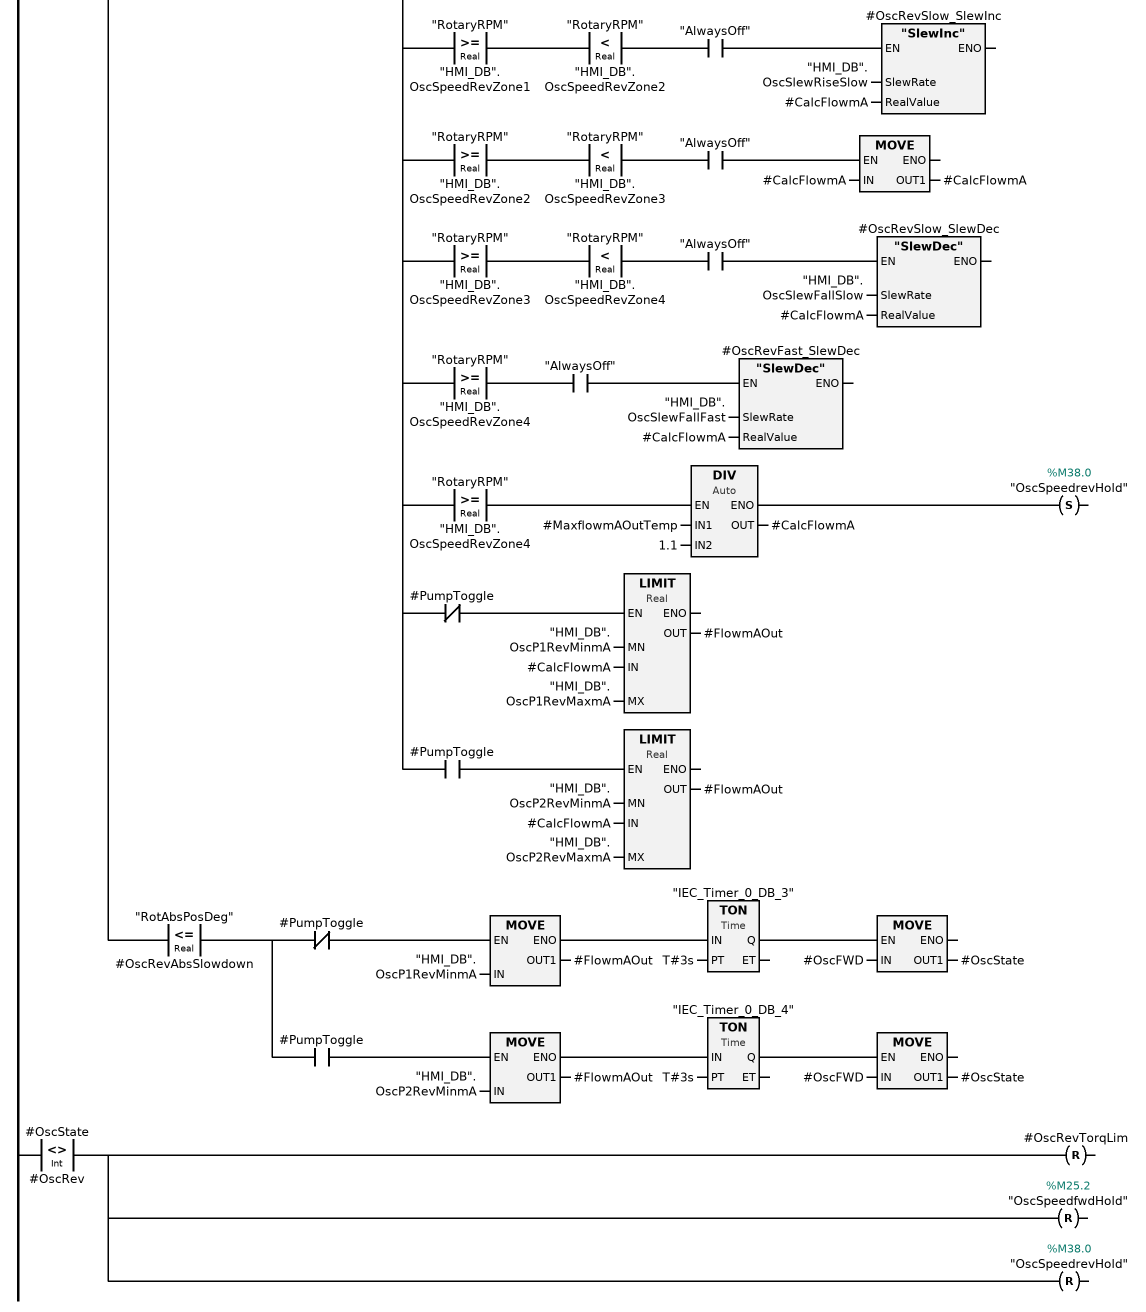
   RUNG wire#powerrail
      { S7_Templates := "SrcType := Int" } EQ_Contact(in1 := #OscState, in2 := #OscRev)
      wire#w1
      P_Trig( #OscRevTrig )
      wire#w2
      I_Contact( #PumpToggle )
      Move(in := "HMI_DB".OscP1HoldmA, out1 => #CalcFlowmA)
   END_RUNG
   RUNG wire#w2
      Contact( #PumpToggle )
      Move(in := "HMI_DB".OscP2HoldmA, out1 => #CalcFlowmA)
   END_RUNG
   RUNG wire#w1
      S_Coil( #FlowRev )
   END_RUNG
   RUNG wire#w1
      { S7_Templates := "SrcType := Real" } GT_Contact(in1 := "RotAbsPosDeg", in2 := #OscRevAbsSlowdown)
      wire#w3
      { S7_Templates := "SrcType := Real" } GE_Contact(in1 := "ActTorqFtLbsFilt", in2 := "HMI_DB".OscTorqRevLowLimFtlbs)
      { S7_Templates := "time_type := Time" } #OscRevTorqLim_TON.TON(pt := "Settings".OscTorqLimTime, et =>)
      S_Coil( #OscRevTorqLim )
   END_RUNG
   RUNG wire#w3
      { S7_Templates := "SrcType := Real" } GE_Contact(in1 := "ActTorqFtLbsFilt", in2 := "HMI_DB".OscTorqRevHighLimFtLbs)
      S_Coil( #OscRevTorqLim )
   END_RUNG
   RUNG wire#w3
      Contact( #OscRevTorqLim )
      P_Trig( #OscRevTorqLimTrig )
      Move(in := #CalcFlowmA, out1 => #LimitFlowmA)
   END_RUNG
   RUNG wire#w3
      { S7_Templates := "SrcType := Real" } LT_Contact(in1 := "ActTorqFtLbsFilt", in2 := "HMI_DB".OscTorqRevLowLimFtlbs)
      { S7_Templates := "SrcType := Real" } LT_Contact(in1 := #CalcFlowmA, in2 := #LimitFlowmA)
      R_Coil( #OscRevTorqLim )
   END_RUNG
   RUNG wire#w3
      Contact( #OscRevTorqLim )
      wire#w4
      { S7_Templates := "SrcType := Real" } GE_Contact(in1 := "ActTorqFtLbsFilt", in2 := "HMI_DB".OscTorqRevHighLimFtLbs)
      Contact( "AlwaysOff" )
      #OscRevTorqLim_SlewDec(SlewRate := "HMI_DB".OscSlewFallSlow, RealValue := #LimitFlowmA)
   END_RUNG
   RUNG wire#w4
      { S7_Templates := "SrcType := Real" } LT_Contact(in1 := "ActTorqFtLbsFilt", in2 := "HMI_DB".OscTorqRevLowLimFtlbs)
      Contact( "AlwaysOff" )
      #OscRevTorqLim_SlewInc(SlewRate := "HMI_DB".OscSlewRiseSlow, RealValue := #LimitFlowmA)
   END_RUNG
   RUNG wire#w4
      I_Contact( #PumpToggle )
      { S7_Templates := "value_type := Real" } Limit(mn := "HMI_DB".OscP1RevMinmA, in := #CalcFlowmA, mx := #LimitFlowmA, out => #CalcFlowmA)
      { S7_Templates := "value_type := Real" } Limit(mn := "HMI_DB".OscP1RevMinmA, in := #CalcFlowmA, mx := "HMI_DB".OscP1RevMaxmA, out => #FlowmAOut)
   END_RUNG
   RUNG wire#w4
      Contact( #PumpToggle )
      { S7_Templates := "value_type := Real" } Limit(mn := "HMI_DB".OscP2RevMinmA, in := #CalcFlowmA, mx := #LimitFlowmA, out => #CalcFlowmA)
      { S7_Templates := "value_type := Real" } Limit(mn := "HMI_DB".OscP2RevMinmA, in := #CalcFlowmA, mx := "HMI_DB".OscP2RevMaxmA, out => #FlowmAOut)
   END_RUNG
   RUNG wire#w3
      I_Contact( #OscRevTorqLim )
      wire#w5
      { S7_Templates := "SrcType := Real" } LT_Contact(in1 := "RotaryRPM", in2 := "HMI_DB".OscSpeedRevZone3)
      I_Contact( "OscSpeedrevHold" )
      #OscRevFast_SlewInc(SlewRate := "HMI_DB".OscSlewRiseFast, RealValue := #CalcFlowmA)
   END_RUNG
   RUNG wire#w5
      { S7_Templates := "SrcType := Real" } GE_Contact(in1 := "RotaryRPM", in2 := "HMI_DB".OscSpeedRevZone1)
      { S7_Templates := "SrcType := Real" } LT_Contact(in1 := "RotaryRPM", in2 := "HMI_DB".OscSpeedRevZone2)
      Contact( "AlwaysOff" )
      #OscRevSlow_SlewInc(SlewRate := "HMI_DB".OscSlewRiseSlow, RealValue := #CalcFlowmA)
   END_RUNG
   RUNG wire#w5
      { S7_Templates := "SrcType := Real" } GE_Contact(in1 := "RotaryRPM", in2 := "HMI_DB".OscSpeedRevZone2)
      { S7_Templates := "SrcType := Real" } LT_Contact(in1 := "RotaryRPM", in2 := "HMI_DB".OscSpeedRevZone3)
      Contact( "AlwaysOff" )
      Move(in := #CalcFlowmA, out1 => #CalcFlowmA)
   END_RUNG
   RUNG wire#w5
      { S7_Templates := "SrcType := Real" } GE_Contact(in1 := "RotaryRPM", in2 := "HMI_DB".OscSpeedRevZone3)
      { S7_Templates := "SrcType := Real" } LT_Contact(in1 := "RotaryRPM", in2 := "HMI_DB".OscSpeedRevZone4)
      Contact( "AlwaysOff" )
      #OscRevSlow_SlewDec(SlewRate := "HMI_DB".OscSlewFallSlow, RealValue := #CalcFlowmA)
   END_RUNG
   RUNG wire#w5
      { S7_Templates := "SrcType := Real" } GE_Contact(in1 := "RotaryRPM", in2 := "HMI_DB".OscSpeedRevZone4)
      Contact( "AlwaysOff" )
      #OscRevFast_SlewDec(SlewRate := "HMI_DB".OscSlewFallFast, RealValue := #CalcFlowmA)
   END_RUNG
   RUNG wire#w5
      { S7_Templates := "SrcType := Real" } GE_Contact(in1 := "RotaryRPM", in2 := "HMI_DB".OscSpeedRevZone4)
      Div(in1 := #MaxflowmAOutTemp, in2 := 1.1, out => #CalcFlowmA)
      S_Coil( "OscSpeedrevHold" )
   END_RUNG
   RUNG wire#w5
      I_Contact( #PumpToggle )
      { S7_Templates := "value_type := Real" } Limit(mn := "HMI_DB".OscP1RevMinmA, in := #CalcFlowmA, mx := "HMI_DB".OscP1RevMaxmA, out => #FlowmAOut)
   END_RUNG
   RUNG wire#w5
      Contact( #PumpToggle )
      { S7_Templates := "value_type := Real" } Limit(mn := "HMI_DB".OscP2RevMinmA, in := #CalcFlowmA, mx := "HMI_DB".OscP2RevMaxmA, out => #FlowmAOut)
   END_RUNG
   RUNG wire#w1
      { S7_Templates := "SrcType := Real" } LE_Contact(in1 := "RotAbsPosDeg", in2 := #OscRevAbsSlowdown)
      wire#w6
      I_Contact( #PumpToggle )
      Move(in := "HMI_DB".OscP1RevMinmA, out1 => #FlowmAOut)
      { S7_Templates := "time_type := Time" } "IEC_Timer_0_DB_3".TON(pt := T#3s, et =>)
      Move(in := #OscFWD, out1 => #OscState)
   END_RUNG
   RUNG wire#w6
      Contact( #PumpToggle )
      Move(in := "HMI_DB".OscP2RevMinmA, out1 => #FlowmAOut)
      { S7_Templates := "time_type := Time" } "IEC_Timer_0_DB_4".TON(pt := T#3s, et =>)
      Move(in := #OscFWD, out1 => #OscState)
   END_RUNG
   RUNG wire#powerrail
      { S7_Templates := "SrcType := Int" } NE_Contact(in1 := #OscState, in2 := #OscRev)
      wire#w7
      R_Coil( #OscRevTorqLim )
   END_RUNG
   RUNG wire#w7
      R_Coil( "OscSpeedfwdHold" )
   END_RUNG
   RUNG wire#w7
      R_Coil( "OscSpeedrevHold" )
   END_RUNG
   // the same network as SCL:
   #_w1 := #OscState = #OscRev;
   #_w2 := #_w1 AND NOT #OscRevTrig;   // rising edge
   #OscRevTrig := #_w1;
   IF #_w2 AND NOT #PumpToggle THEN #CalcFlowmA := "HMI_DB".OscP1HoldmA; END_IF;
   IF #_w2 AND #PumpToggle THEN #CalcFlowmA := "HMI_DB".OscP2HoldmA; END_IF;
   IF #_w1 THEN #FlowRev := TRUE; END_IF;
   #_w3 := #_w1 AND ("RotAbsPosDeg" > #OscRevAbsSlowdown);
   #OscRevTorqLim_TON(IN := #_w3 AND ("ActTorqFtLbsFilt" >= "HMI_DB".OscTorqRevLowLimFtlbs),   // TON
                      PT := "Settings".OscTorqLimTime);
   IF #OscRevTorqLim_TON.Q THEN #OscRevTorqLim := TRUE; END_IF;
   IF #_w3 AND ("ActTorqFtLbsFilt" >= "HMI_DB".OscTorqRevHighLimFtLbs) THEN #OscRevTorqLim := TRUE; END_IF;
   #_w4 := #_w3 AND #OscRevTorqLim;
   #_w5 := #_w4 AND NOT #OscRevTorqLimTrig;   // rising edge
   #OscRevTorqLimTrig := #_w4;
   IF #_w5 THEN #LimitFlowmA := #CalcFlowmA; END_IF;
   IF #_w3 AND ("ActTorqFtLbsFilt" < "HMI_DB".OscTorqRevLowLimFtlbs) AND (#CalcFlowmA < #LimitFlowmA) THEN
       #OscRevTorqLim := FALSE;
   END_IF;
   #_w6 := #_w3 AND #OscRevTorqLim;
   IF #_w6 AND ("ActTorqFtLbsFilt" >= "HMI_DB".OscTorqRevHighLimFtLbs) AND "AlwaysOff" THEN
       #OscRevTorqLim_SlewDec(SlewRate := "HMI_DB".OscSlewFallSlow, RealValue := #LimitFlowmA);   // "SlewDec"
   END_IF;
   IF #_w6 AND ("ActTorqFtLbsFilt" < "HMI_DB".OscTorqRevLowLimFtlbs) AND "AlwaysOff" THEN
       #OscRevTorqLim_SlewInc(SlewRate := "HMI_DB".OscSlewRiseSlow, RealValue := #LimitFlowmA);   // "SlewInc"
   END_IF;
   IF #_w6 AND NOT #PumpToggle THEN
       #CalcFlowmA := LIMIT(MN := "HMI_DB".OscP1RevMinmA, IN := #CalcFlowmA, MX := #LimitFlowmA);
       #FlowmAOut := LIMIT(MN := "HMI_DB".OscP1RevMinmA, IN := #CalcFlowmA, MX := "HMI_DB".OscP1RevMaxmA);
   END_IF;
   IF #_w6 AND #PumpToggle THEN
       #CalcFlowmA := LIMIT(MN := "HMI_DB".OscP2RevMinmA, IN := #CalcFlowmA, MX := #LimitFlowmA);
       #FlowmAOut := LIMIT(MN := "HMI_DB".OscP2RevMinmA, IN := #CalcFlowmA, MX := "HMI_DB".OscP2RevMaxmA);
   END_IF;
   #_w7 := #_w3 AND NOT #OscRevTorqLim;
   IF #_w7 AND ("RotaryRPM" < "HMI_DB".OscSpeedRevZone3) AND NOT "OscSpeedrevHold" THEN
       #OscRevFast_SlewInc(SlewRate := "HMI_DB".OscSlewRiseFast, RealValue := #CalcFlowmA);   // "SlewInc"
   END_IF;
   IF #_w7 AND ("RotaryRPM" >= "HMI_DB".OscSpeedRevZone1) AND ("RotaryRPM" < "HMI_DB".OscSpeedRevZone2) AND "AlwaysOff" THEN
       #OscRevSlow_SlewInc(SlewRate := "HMI_DB".OscSlewRiseSlow, RealValue := #CalcFlowmA);   // "SlewInc"
   END_IF;
   IF #_w7 AND ("RotaryRPM" >= "HMI_DB".OscSpeedRevZone2) AND ("RotaryRPM" < "HMI_DB".OscSpeedRevZone3) AND "AlwaysOff" THEN
       #CalcFlowmA := #CalcFlowmA;
   END_IF;
   IF #_w7 AND ("RotaryRPM" >= "HMI_DB".OscSpeedRevZone3) AND ("RotaryRPM" < "HMI_DB".OscSpeedRevZone4) AND "AlwaysOff" THEN
       #OscRevSlow_SlewDec(SlewRate := "HMI_DB".OscSlewFallSlow, RealValue := #CalcFlowmA);   // "SlewDec"
   END_IF;
   IF #_w7 AND ("RotaryRPM" >= "HMI_DB".OscSpeedRevZone4) AND "AlwaysOff" THEN
       #OscRevFast_SlewDec(SlewRate := "HMI_DB".OscSlewFallFast, RealValue := #CalcFlowmA);   // "SlewDec"
   END_IF;
   IF #_w7 AND ("RotaryRPM" >= "HMI_DB".OscSpeedRevZone4) THEN
       #CalcFlowmA := #MaxflowmAOutTemp / 1.1;
       "OscSpeedrevHold" := TRUE;
   END_IF;
   IF #_w7 AND NOT #PumpToggle THEN
       #FlowmAOut := LIMIT(MN := "HMI_DB".OscP1RevMinmA, IN := #CalcFlowmA, MX := "HMI_DB".OscP1RevMaxmA);
   END_IF;
   IF #_w7 AND #PumpToggle THEN
       #FlowmAOut := LIMIT(MN := "HMI_DB".OscP2RevMinmA, IN := #CalcFlowmA, MX := "HMI_DB".OscP2RevMaxmA);
   END_IF;
   #_w8 := #_w1 AND ("RotAbsPosDeg" <= #OscRevAbsSlowdown);
   #_w9 := #_w8 AND NOT #PumpToggle;
   IF #_w9 THEN #FlowmAOut := "HMI_DB".OscP1RevMinmA; END_IF;
   "IEC_Timer_0_DB_3".TON(IN := #_w9, PT := T#3s);
   IF "IEC_Timer_0_DB_3".Q THEN #OscState := #OscFWD; END_IF;
   #_w10 := #_w8 AND #PumpToggle;
   IF #_w10 THEN #FlowmAOut := "HMI_DB".OscP2RevMinmA; END_IF;
   "IEC_Timer_0_DB_4".TON(IN := #_w10, PT := T#3s);
   IF "IEC_Timer_0_DB_4".Q THEN #OscState := #OscFWD; END_IF;
   IF #OscState <> #OscRev THEN
       #OscRevTorqLim := FALSE;
       "OscSpeedfwdHold" := FALSE;
       "OscSpeedrevHold" := FALSE;
   END_IF;
END_REGION

REGION Network 16: Stop Oscillating - State 250
   // Determine current position and direction to Home position
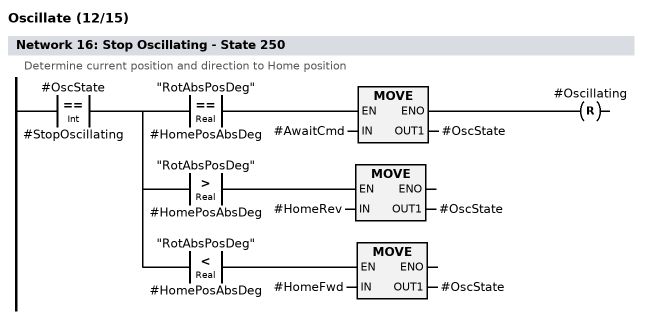
   RUNG wire#powerrail
      { S7_Templates := "SrcType := Int" } EQ_Contact(in1 := #OscState, in2 := #StopOscillating)
      wire#w1
      { S7_Templates := "SrcType := Real" } EQ_Contact(in1 := "RotAbsPosDeg", in2 := #HomePosAbsDeg)
      Move(in := #AwaitCmd, out1 => #OscState)
      R_Coil( #Oscillating )
   END_RUNG
   RUNG wire#w1
      { S7_Templates := "SrcType := Real" } GT_Contact(in1 := "RotAbsPosDeg", in2 := #HomePosAbsDeg)
      Move(in := #HomeRev, out1 => #OscState)
   END_RUNG
   RUNG wire#w1
      { S7_Templates := "SrcType := Real" } LT_Contact(in1 := "RotAbsPosDeg", in2 := #HomePosAbsDeg)
      Move(in := #HomeFwd, out1 => #OscState)
   END_RUNG
   // the same network as SCL:
   #_w1 := #OscState = #StopOscillating;
   IF #_w1 AND ("RotAbsPosDeg" = #HomePosAbsDeg) THEN
       #OscState := #AwaitCmd;
       #Oscillating := FALSE;
   END_IF;
   IF #_w1 AND ("RotAbsPosDeg" > #HomePosAbsDeg) THEN #OscState := #HomeRev; END_IF;
   IF #_w1 AND ("RotAbsPosDeg" < #HomePosAbsDeg) THEN #OscState := #HomeFwd; END_IF;
END_REGION

REGION Network 17: Home Fwd - State 251
   // Move quill FWD to the home position
   // Start at Min and Ramp up until speed reach. 
   // If Approaching Torq Limit, limit output flow. 
   // At or above end position, switch direction
   // Note: Dummy Move On Maintain speed there as visual only.
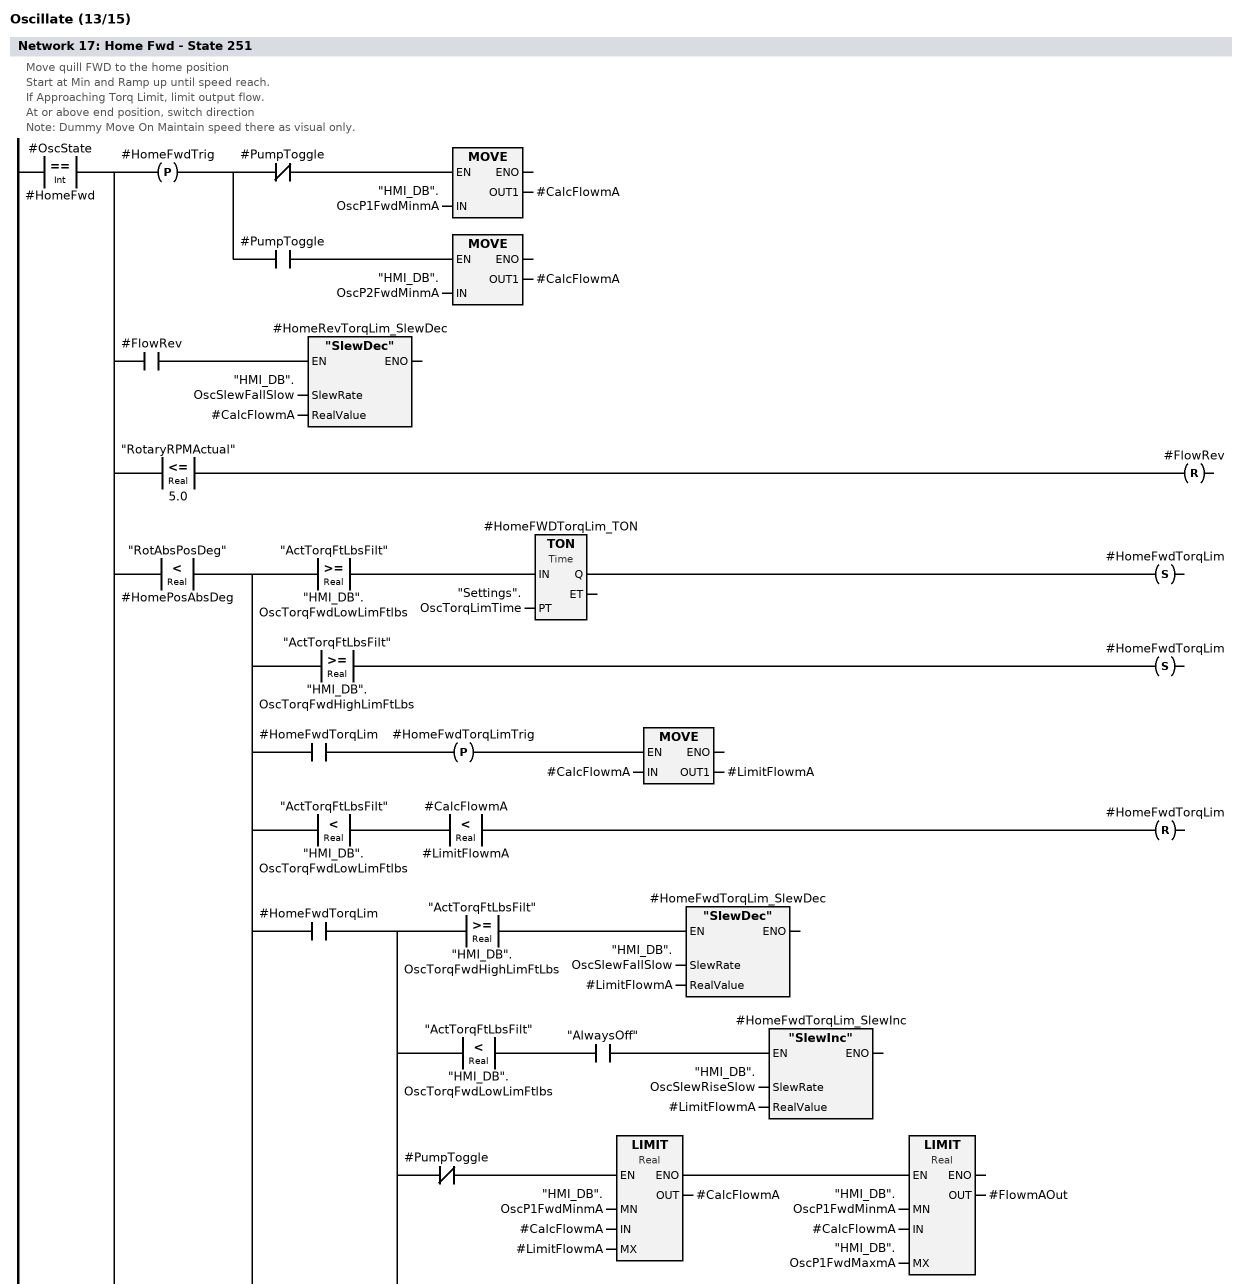
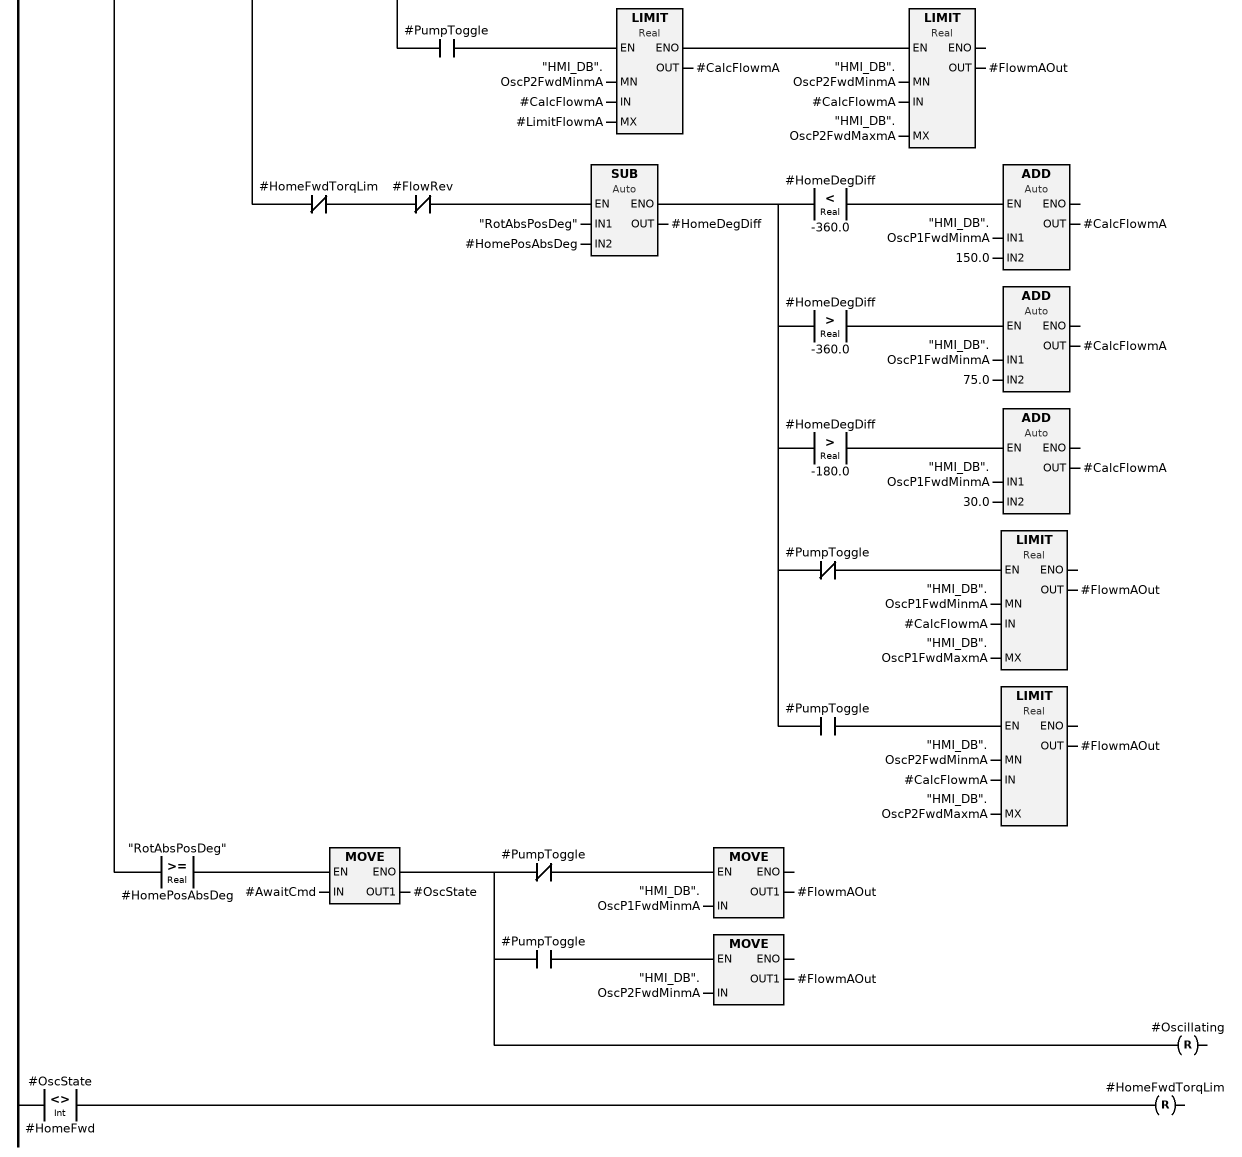
   RUNG wire#powerrail
      { S7_Templates := "SrcType := Int" } EQ_Contact(in1 := #OscState, in2 := #HomeFwd)
      wire#w1
      P_Trig( #HomeFwdTrig )
      wire#w2
      I_Contact( #PumpToggle )
      Move(in := "HMI_DB".OscP1FwdMinmA, out1 => #CalcFlowmA)
   END_RUNG
   RUNG wire#w2
      Contact( #PumpToggle )
      Move(in := "HMI_DB".OscP2FwdMinmA, out1 => #CalcFlowmA)
   END_RUNG
   RUNG wire#w1
      Contact( #FlowRev )
      #HomeRevTorqLim_SlewDec(SlewRate := "HMI_DB".OscSlewFallSlow, RealValue := #CalcFlowmA)
   END_RUNG
   RUNG wire#w1
      { S7_Templates := "SrcType := Real" } LE_Contact(in1 := "RotaryRPMActual", in2 := 5.0)
      R_Coil( #FlowRev )
   END_RUNG
   RUNG wire#w1
      { S7_Templates := "SrcType := Real" } LT_Contact(in1 := "RotAbsPosDeg", in2 := #HomePosAbsDeg)
      wire#w3
      { S7_Templates := "SrcType := Real" } GE_Contact(in1 := "ActTorqFtLbsFilt", in2 := "HMI_DB".OscTorqFwdLowLimFtlbs)
      { S7_Templates := "time_type := Time" } #HomeFWDTorqLim_TON.TON(pt := "Settings".OscTorqLimTime, et =>)
      S_Coil( #HomeFwdTorqLim )
   END_RUNG
   RUNG wire#w3
      { S7_Templates := "SrcType := Real" } GE_Contact(in1 := "ActTorqFtLbsFilt", in2 := "HMI_DB".OscTorqFwdHighLimFtLbs)
      S_Coil( #HomeFwdTorqLim )
   END_RUNG
   RUNG wire#w3
      Contact( #HomeFwdTorqLim )
      P_Trig( #HomeFwdTorqLimTrig )
      Move(in := #CalcFlowmA, out1 => #LimitFlowmA)
   END_RUNG
   RUNG wire#w3
      { S7_Templates := "SrcType := Real" } LT_Contact(in1 := "ActTorqFtLbsFilt", in2 := "HMI_DB".OscTorqFwdLowLimFtlbs)
      { S7_Templates := "SrcType := Real" } LT_Contact(in1 := #CalcFlowmA, in2 := #LimitFlowmA)
      R_Coil( #HomeFwdTorqLim )
   END_RUNG
   RUNG wire#w3
      Contact( #HomeFwdTorqLim )
      wire#w4
      { S7_Templates := "SrcType := Real" } GE_Contact(in1 := "ActTorqFtLbsFilt", in2 := "HMI_DB".OscTorqFwdHighLimFtLbs)
      #HomeFwdTorqLim_SlewDec(SlewRate := "HMI_DB".OscSlewFallSlow, RealValue := #LimitFlowmA)
   END_RUNG
   RUNG wire#w4
      { S7_Templates := "SrcType := Real" } LT_Contact(in1 := "ActTorqFtLbsFilt", in2 := "HMI_DB".OscTorqFwdLowLimFtlbs)
      Contact( "AlwaysOff" )
      #HomeFwdTorqLim_SlewInc(SlewRate := "HMI_DB".OscSlewRiseSlow, RealValue := #LimitFlowmA)
   END_RUNG
   RUNG wire#w4
      I_Contact( #PumpToggle )
      { S7_Templates := "value_type := Real" } Limit(mn := "HMI_DB".OscP1FwdMinmA, in := #CalcFlowmA, mx := #LimitFlowmA, out => #CalcFlowmA)
      { S7_Templates := "value_type := Real" } Limit(mn := "HMI_DB".OscP1FwdMinmA, in := #CalcFlowmA, mx := "HMI_DB".OscP1FwdMaxmA, out => #FlowmAOut)
   END_RUNG
   RUNG wire#w4
      Contact( #PumpToggle )
      { S7_Templates := "value_type := Real" } Limit(mn := "HMI_DB".OscP2FwdMinmA, in := #CalcFlowmA, mx := #LimitFlowmA, out => #CalcFlowmA)
      { S7_Templates := "value_type := Real" } Limit(mn := "HMI_DB".OscP2FwdMinmA, in := #CalcFlowmA, mx := "HMI_DB".OscP2FwdMaxmA, out => #FlowmAOut)
   END_RUNG
   RUNG wire#w3
      I_Contact( #HomeFwdTorqLim )
      I_Contact( #FlowRev )
      Sub(in1 := "RotAbsPosDeg", in2 := #HomePosAbsDeg, out => #HomeDegDiff)
      wire#w5
      { S7_Templates := "SrcType := Real" } LT_Contact(in1 := #HomeDegDiff, in2 := -360.0)
      Add(in1 := "HMI_DB".OscP1FwdMinmA, in2 := 150.0, out => #CalcFlowmA)
   END_RUNG
   RUNG wire#w5
      { S7_Templates := "SrcType := Real" } GT_Contact(in1 := #HomeDegDiff, in2 := -360.0)
      Add(in1 := "HMI_DB".OscP1FwdMinmA, in2 := 75.0, out => #CalcFlowmA)
   END_RUNG
   RUNG wire#w5
      { S7_Templates := "SrcType := Real" } GT_Contact(in1 := #HomeDegDiff, in2 := -180.0)
      Add(in1 := "HMI_DB".OscP1FwdMinmA, in2 := 30.0, out => #CalcFlowmA)
   END_RUNG
   RUNG wire#w5
      I_Contact( #PumpToggle )
      { S7_Templates := "value_type := Real" } Limit(mn := "HMI_DB".OscP1FwdMinmA, in := #CalcFlowmA, mx := "HMI_DB".OscP1FwdMaxmA, out => #FlowmAOut)
   END_RUNG
   RUNG wire#w5
      Contact( #PumpToggle )
      { S7_Templates := "value_type := Real" } Limit(mn := "HMI_DB".OscP2FwdMinmA, in := #CalcFlowmA, mx := "HMI_DB".OscP2FwdMaxmA, out => #FlowmAOut)
   END_RUNG
   RUNG wire#w1
      { S7_Templates := "SrcType := Real" } GE_Contact(in1 := "RotAbsPosDeg", in2 := #HomePosAbsDeg)
      Move(in := #AwaitCmd, out1 => #OscState)
      wire#w6
      I_Contact( #PumpToggle )
      Move(in := "HMI_DB".OscP1FwdMinmA, out1 => #FlowmAOut)
   END_RUNG
   RUNG wire#w6
      Contact( #PumpToggle )
      Move(in := "HMI_DB".OscP2FwdMinmA, out1 => #FlowmAOut)
   END_RUNG
   RUNG wire#w6
      R_Coil( #Oscillating )
   END_RUNG
   RUNG wire#powerrail
      { S7_Templates := "SrcType := Int" } NE_Contact(in1 := #OscState, in2 := #HomeFwd)
      R_Coil( #HomeFwdTorqLim )
   END_RUNG
   // the same network as SCL:
   #_w1 := #OscState = #HomeFwd;
   #_w2 := #_w1 AND NOT #HomeFwdTrig;   // rising edge
   #HomeFwdTrig := #_w1;
   IF #_w2 AND NOT #PumpToggle THEN #CalcFlowmA := "HMI_DB".OscP1FwdMinmA; END_IF;
   IF #_w2 AND #PumpToggle THEN #CalcFlowmA := "HMI_DB".OscP2FwdMinmA; END_IF;
   IF #_w1 AND #FlowRev THEN
       #HomeRevTorqLim_SlewDec(SlewRate := "HMI_DB".OscSlewFallSlow, RealValue := #CalcFlowmA);   // "SlewDec"
   END_IF;
   IF #_w1 AND ("RotaryRPMActual" <= 5.0) THEN #FlowRev := FALSE; END_IF;
   #_w3 := #_w1 AND ("RotAbsPosDeg" < #HomePosAbsDeg);
   #HomeFWDTorqLim_TON(IN := #_w3 AND ("ActTorqFtLbsFilt" >= "HMI_DB".OscTorqFwdLowLimFtlbs),   // TON
                       PT := "Settings".OscTorqLimTime);
   IF #HomeFWDTorqLim_TON.Q THEN #HomeFwdTorqLim := TRUE; END_IF;
   IF #_w3 AND ("ActTorqFtLbsFilt" >= "HMI_DB".OscTorqFwdHighLimFtLbs) THEN #HomeFwdTorqLim := TRUE; END_IF;
   #_w4 := #_w3 AND #HomeFwdTorqLim;
   #_w5 := #_w4 AND NOT #HomeFwdTorqLimTrig;   // rising edge
   #HomeFwdTorqLimTrig := #_w4;
   IF #_w5 THEN #LimitFlowmA := #CalcFlowmA; END_IF;
   IF #_w3 AND ("ActTorqFtLbsFilt" < "HMI_DB".OscTorqFwdLowLimFtlbs) AND (#CalcFlowmA < #LimitFlowmA) THEN
       #HomeFwdTorqLim := FALSE;
   END_IF;
   #_w6 := #_w3 AND #HomeFwdTorqLim;
   IF #_w6 AND ("ActTorqFtLbsFilt" >= "HMI_DB".OscTorqFwdHighLimFtLbs) THEN
       #HomeFwdTorqLim_SlewDec(SlewRate := "HMI_DB".OscSlewFallSlow, RealValue := #LimitFlowmA);   // "SlewDec"
   END_IF;
   IF #_w6 AND ("ActTorqFtLbsFilt" < "HMI_DB".OscTorqFwdLowLimFtlbs) AND "AlwaysOff" THEN
       #HomeFwdTorqLim_SlewInc(SlewRate := "HMI_DB".OscSlewRiseSlow, RealValue := #LimitFlowmA);   // "SlewInc"
   END_IF;
   IF #_w6 AND NOT #PumpToggle THEN
       #CalcFlowmA := LIMIT(MN := "HMI_DB".OscP1FwdMinmA, IN := #CalcFlowmA, MX := #LimitFlowmA);
       #FlowmAOut := LIMIT(MN := "HMI_DB".OscP1FwdMinmA, IN := #CalcFlowmA, MX := "HMI_DB".OscP1FwdMaxmA);
   END_IF;
   IF #_w6 AND #PumpToggle THEN
       #CalcFlowmA := LIMIT(MN := "HMI_DB".OscP2FwdMinmA, IN := #CalcFlowmA, MX := #LimitFlowmA);
       #FlowmAOut := LIMIT(MN := "HMI_DB".OscP2FwdMinmA, IN := #CalcFlowmA, MX := "HMI_DB".OscP2FwdMaxmA);
   END_IF;
   #_w7 := #_w3 AND NOT #HomeFwdTorqLim AND NOT #FlowRev;
   IF #_w7 THEN #HomeDegDiff := "RotAbsPosDeg" - #HomePosAbsDeg; END_IF;
   IF #_w7 AND (#HomeDegDiff < (-360.0)) THEN #CalcFlowmA := "HMI_DB".OscP1FwdMinmA + 150.0; END_IF;
   IF #_w7 AND (#HomeDegDiff > (-360.0)) THEN #CalcFlowmA := "HMI_DB".OscP1FwdMinmA + 75.0; END_IF;
   IF #_w7 AND (#HomeDegDiff > (-180.0)) THEN #CalcFlowmA := "HMI_DB".OscP1FwdMinmA + 30.0; END_IF;
   IF #_w7 AND NOT #PumpToggle THEN
       #FlowmAOut := LIMIT(MN := "HMI_DB".OscP1FwdMinmA, IN := #CalcFlowmA, MX := "HMI_DB".OscP1FwdMaxmA);
   END_IF;
   IF #_w7 AND #PumpToggle THEN
       #FlowmAOut := LIMIT(MN := "HMI_DB".OscP2FwdMinmA, IN := #CalcFlowmA, MX := "HMI_DB".OscP2FwdMaxmA);
   END_IF;
   #_w8 := #_w1 AND ("RotAbsPosDeg" >= #HomePosAbsDeg);
   IF #_w8 THEN #OscState := #AwaitCmd; END_IF;
   IF #_w8 AND NOT #PumpToggle THEN #FlowmAOut := "HMI_DB".OscP1FwdMinmA; END_IF;
   IF #_w8 AND #PumpToggle THEN #FlowmAOut := "HMI_DB".OscP2FwdMinmA; END_IF;
   IF #_w8 THEN #Oscillating := FALSE; END_IF;
   IF #OscState <> #HomeFwd THEN #HomeFwdTorqLim := FALSE; END_IF;
END_REGION

REGION Network 18: Home Rev - State 252
   // Move quill to Home position in the Rev direction. 
   // Start at Hold mA and Ramp up until speed reach. 
   // If Approaching Torq Limit, limit output flow. 
   // At or above new home position, output hold value and hold position
   // Note: Dummy Move On Maintain speed there as visual only.
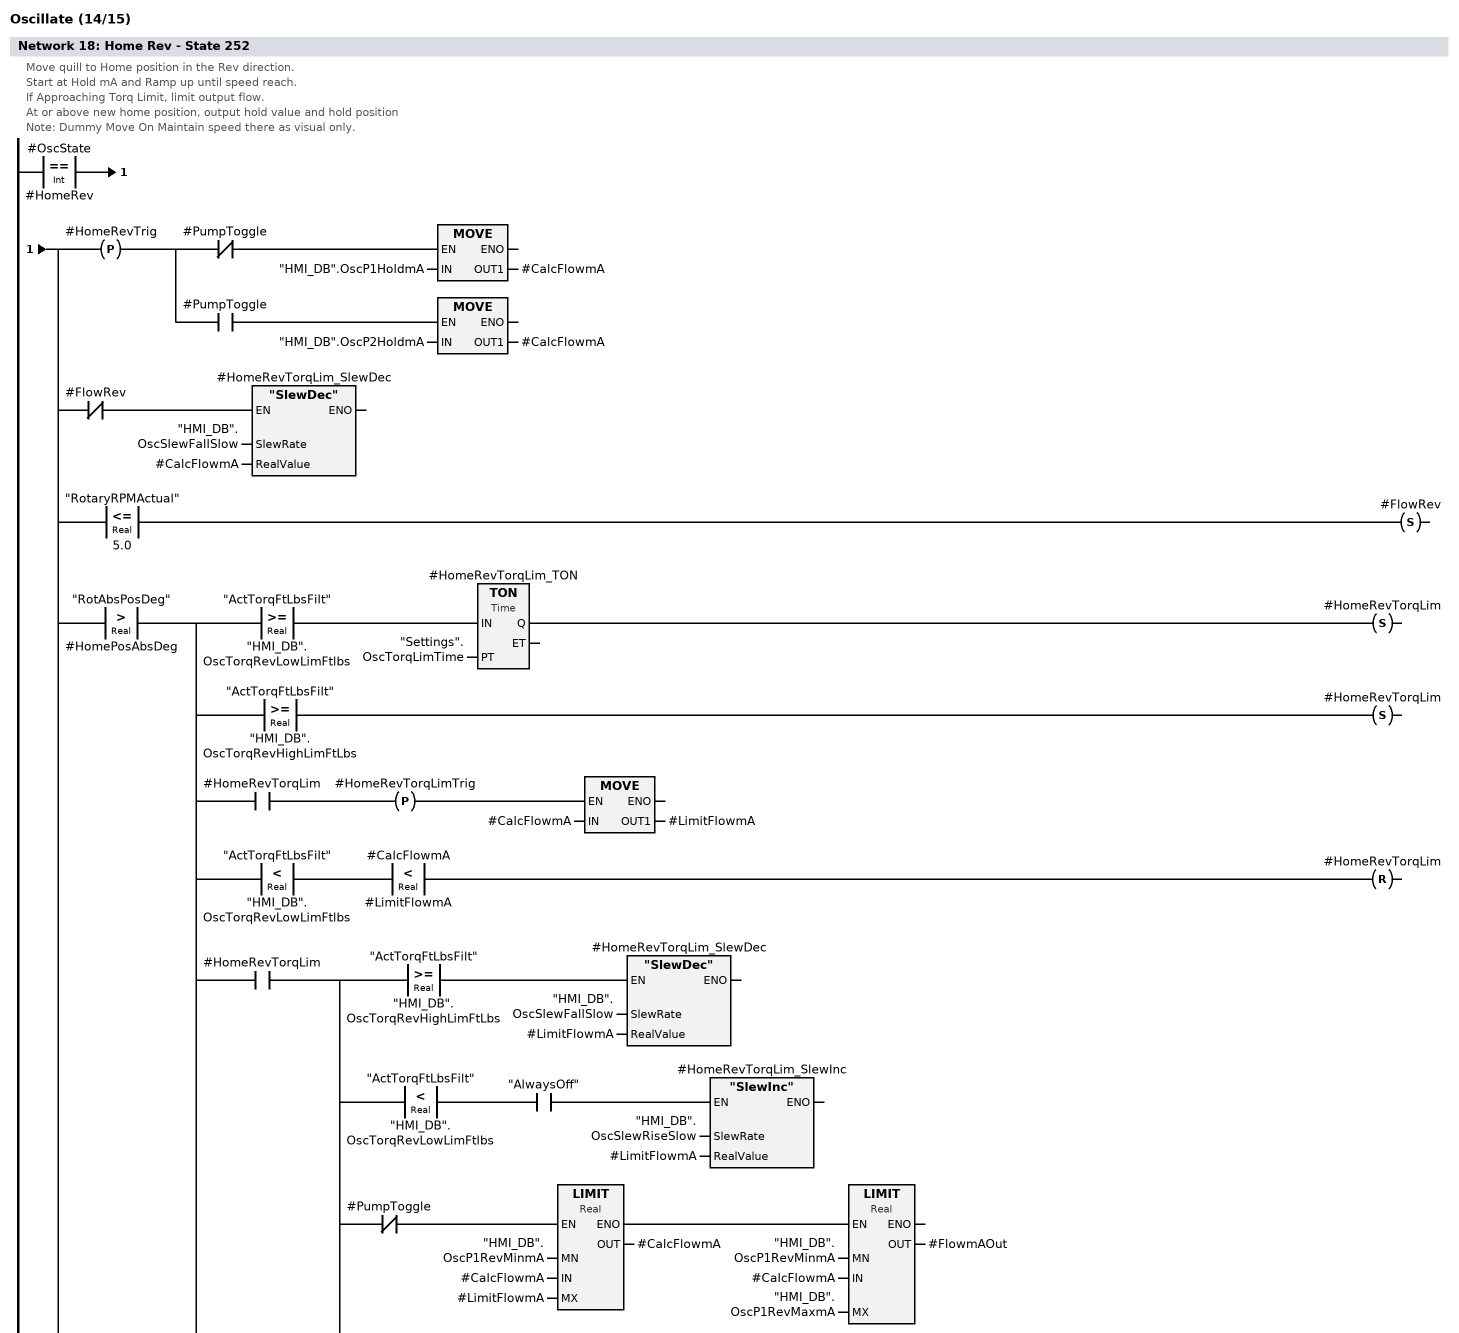
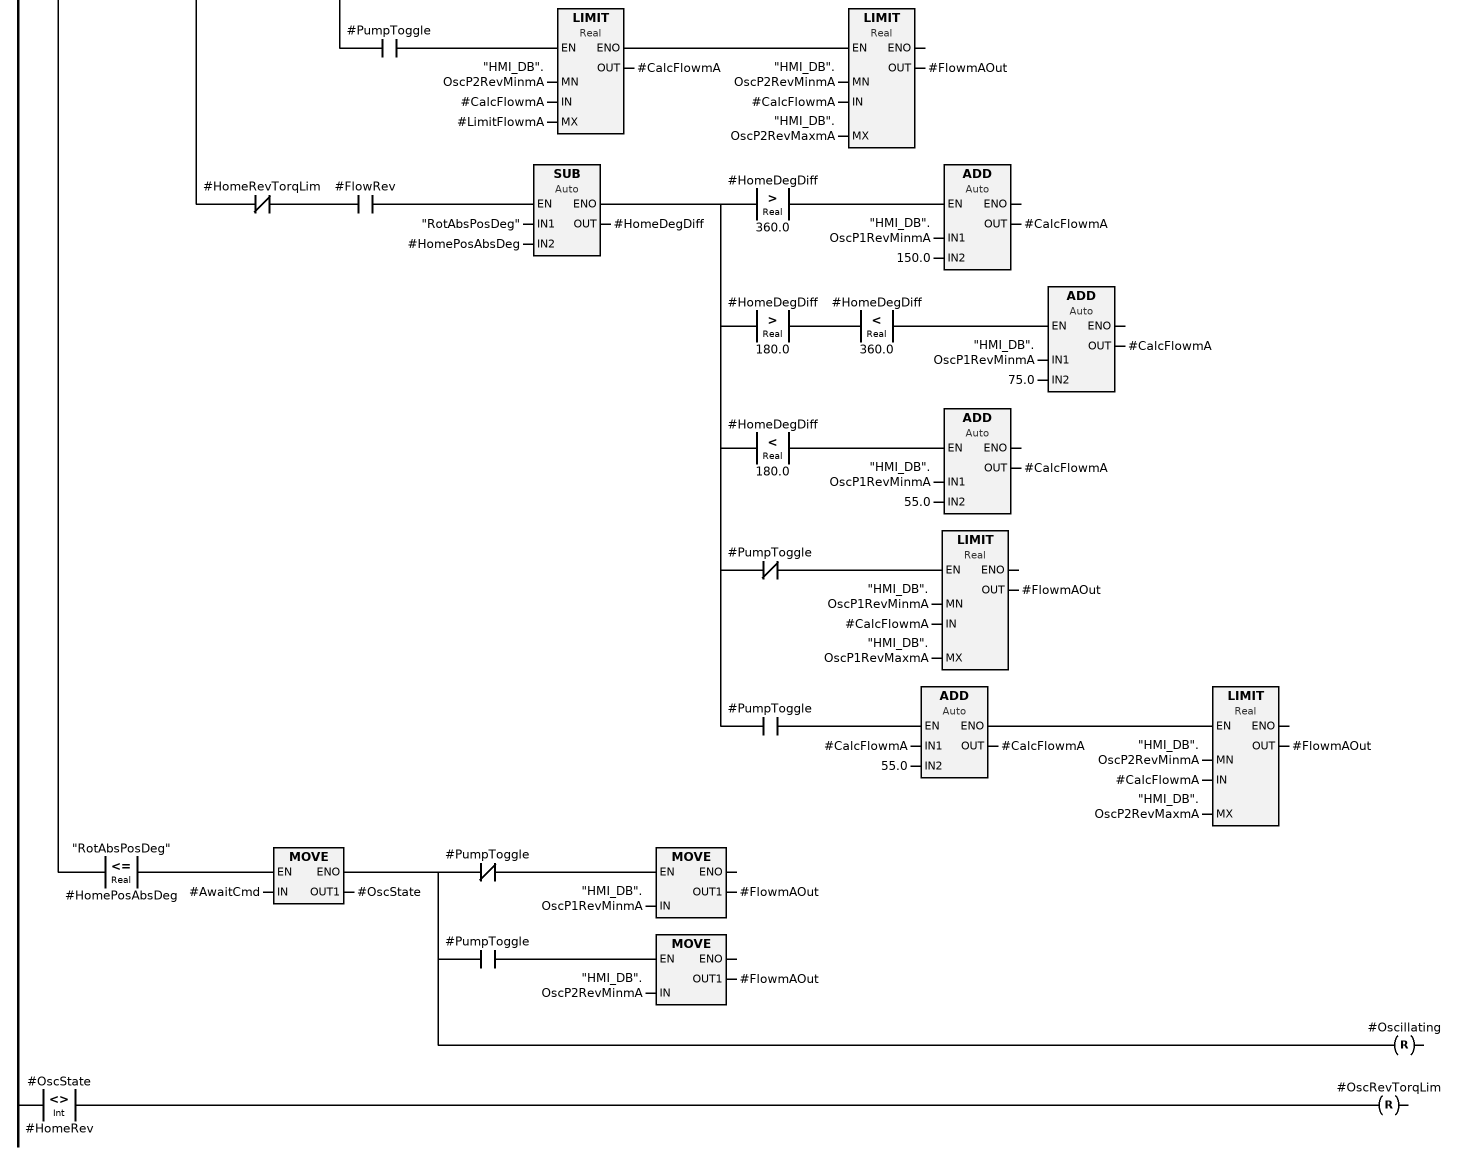
   RUNG wire#powerrail
      { S7_Templates := "SrcType := Int" } EQ_Contact(in1 := #OscState, in2 := #HomeRev)
      wire#w1
      P_Trig( #HomeRevTrig )
      wire#w2
      I_Contact( #PumpToggle )
      Move(in := "HMI_DB".OscP1HoldmA, out1 => #CalcFlowmA)
   END_RUNG
   RUNG wire#w2
      Contact( #PumpToggle )
      Move(in := "HMI_DB".OscP2HoldmA, out1 => #CalcFlowmA)
   END_RUNG
   RUNG wire#w1
      I_Contact( #FlowRev )
      #HomeRevTorqLim_SlewDec(SlewRate := "HMI_DB".OscSlewFallSlow, RealValue := #CalcFlowmA)
   END_RUNG
   RUNG wire#w1
      { S7_Templates := "SrcType := Real" } LE_Contact(in1 := "RotaryRPMActual", in2 := 5.0)
      S_Coil( #FlowRev )
   END_RUNG
   RUNG wire#w1
      { S7_Templates := "SrcType := Real" } GT_Contact(in1 := "RotAbsPosDeg", in2 := #HomePosAbsDeg)
      wire#w3
      { S7_Templates := "SrcType := Real" } GE_Contact(in1 := "ActTorqFtLbsFilt", in2 := "HMI_DB".OscTorqRevLowLimFtlbs)
      { S7_Templates := "time_type := Time" } #HomeRevTorqLim_TON.TON(pt := "Settings".OscTorqLimTime, et =>)
      S_Coil( #HomeRevTorqLim )
   END_RUNG
   RUNG wire#w3
      { S7_Templates := "SrcType := Real" } GE_Contact(in1 := "ActTorqFtLbsFilt", in2 := "HMI_DB".OscTorqRevHighLimFtLbs)
      S_Coil( #HomeRevTorqLim )
   END_RUNG
   RUNG wire#w3
      Contact( #HomeRevTorqLim )
      P_Trig( #HomeRevTorqLimTrig )
      Move(in := #CalcFlowmA, out1 => #LimitFlowmA)
   END_RUNG
   RUNG wire#w3
      { S7_Templates := "SrcType := Real" } LT_Contact(in1 := "ActTorqFtLbsFilt", in2 := "HMI_DB".OscTorqRevLowLimFtlbs)
      { S7_Templates := "SrcType := Real" } LT_Contact(in1 := #CalcFlowmA, in2 := #LimitFlowmA)
      R_Coil( #HomeRevTorqLim )
   END_RUNG
   RUNG wire#w3
      Contact( #HomeRevTorqLim )
      wire#w4
      { S7_Templates := "SrcType := Real" } GE_Contact(in1 := "ActTorqFtLbsFilt", in2 := "HMI_DB".OscTorqRevHighLimFtLbs)
      #HomeRevTorqLim_SlewDec(SlewRate := "HMI_DB".OscSlewFallSlow, RealValue := #LimitFlowmA)
   END_RUNG
   RUNG wire#w4
      { S7_Templates := "SrcType := Real" } LT_Contact(in1 := "ActTorqFtLbsFilt", in2 := "HMI_DB".OscTorqRevLowLimFtlbs)
      Contact( "AlwaysOff" )
      #HomeRevTorqLim_SlewInc(SlewRate := "HMI_DB".OscSlewRiseSlow, RealValue := #LimitFlowmA)
   END_RUNG
   RUNG wire#w4
      I_Contact( #PumpToggle )
      { S7_Templates := "value_type := Real" } Limit(mn := "HMI_DB".OscP1RevMinmA, in := #CalcFlowmA, mx := #LimitFlowmA, out => #CalcFlowmA)
      { S7_Templates := "value_type := Real" } Limit(mn := "HMI_DB".OscP1RevMinmA, in := #CalcFlowmA, mx := "HMI_DB".OscP1RevMaxmA, out => #FlowmAOut)
   END_RUNG
   RUNG wire#w4
      Contact( #PumpToggle )
      { S7_Templates := "value_type := Real" } Limit(mn := "HMI_DB".OscP2RevMinmA, in := #CalcFlowmA, mx := #LimitFlowmA, out => #CalcFlowmA)
      { S7_Templates := "value_type := Real" } Limit(mn := "HMI_DB".OscP2RevMinmA, in := #CalcFlowmA, mx := "HMI_DB".OscP2RevMaxmA, out => #FlowmAOut)
   END_RUNG
   RUNG wire#w3
      I_Contact( #HomeRevTorqLim )
      Contact( #FlowRev )
      Sub(in1 := "RotAbsPosDeg", in2 := #HomePosAbsDeg, out => #HomeDegDiff)
      wire#w5
      { S7_Templates := "SrcType := Real" } GT_Contact(in1 := #HomeDegDiff, in2 := 360.0)
      Add(in1 := "HMI_DB".OscP1RevMinmA, in2 := 150.0, out => #CalcFlowmA)
   END_RUNG
   RUNG wire#w5
      { S7_Templates := "SrcType := Real" } GT_Contact(in1 := #HomeDegDiff, in2 := 180.0)
      { S7_Templates := "SrcType := Real" } LT_Contact(in1 := #HomeDegDiff, in2 := 360.0)
      Add(in1 := "HMI_DB".OscP1RevMinmA, in2 := 75.0, out => #CalcFlowmA)
   END_RUNG
   RUNG wire#w5
      { S7_Templates := "SrcType := Real" } LT_Contact(in1 := #HomeDegDiff, in2 := 180.0)
      Add(in1 := "HMI_DB".OscP1RevMinmA, in2 := 55.0, out => #CalcFlowmA)
   END_RUNG
   RUNG wire#w5
      I_Contact( #PumpToggle )
      { S7_Templates := "value_type := Real" } Limit(mn := "HMI_DB".OscP1RevMinmA, in := #CalcFlowmA, mx := "HMI_DB".OscP1RevMaxmA, out => #FlowmAOut)
   END_RUNG
   RUNG wire#w5
      Contact( #PumpToggle )
      Add(in1 := #CalcFlowmA, in2 := 55.0, out => #CalcFlowmA)
      { S7_Templates := "value_type := Real" } Limit(mn := "HMI_DB".OscP2RevMinmA, in := #CalcFlowmA, mx := "HMI_DB".OscP2RevMaxmA, out => #FlowmAOut)
   END_RUNG
   RUNG wire#w1
      { S7_Templates := "SrcType := Real" } LE_Contact(in1 := "RotAbsPosDeg", in2 := #HomePosAbsDeg)
      Move(in := #AwaitCmd, out1 => #OscState)
      wire#w6
      I_Contact( #PumpToggle )
      Move(in := "HMI_DB".OscP1RevMinmA, out1 => #FlowmAOut)
   END_RUNG
   RUNG wire#w6
      Contact( #PumpToggle )
      Move(in := "HMI_DB".OscP2RevMinmA, out1 => #FlowmAOut)
   END_RUNG
   RUNG wire#w6
      R_Coil( #Oscillating )
   END_RUNG
   RUNG wire#powerrail
      { S7_Templates := "SrcType := Int" } NE_Contact(in1 := #OscState, in2 := #HomeRev)
      R_Coil( #OscRevTorqLim )
   END_RUNG
   // the same network as SCL:
   #_w1 := #OscState = #HomeRev;
   #_w2 := #_w1 AND NOT #HomeRevTrig;   // rising edge
   #HomeRevTrig := #_w1;
   IF #_w2 AND NOT #PumpToggle THEN #CalcFlowmA := "HMI_DB".OscP1HoldmA; END_IF;
   IF #_w2 AND #PumpToggle THEN #CalcFlowmA := "HMI_DB".OscP2HoldmA; END_IF;
   IF #_w1 AND NOT #FlowRev THEN
       #HomeRevTorqLim_SlewDec(SlewRate := "HMI_DB".OscSlewFallSlow, RealValue := #CalcFlowmA);   // "SlewDec"
   END_IF;
   IF #_w1 AND ("RotaryRPMActual" <= 5.0) THEN #FlowRev := TRUE; END_IF;
   #_w3 := #_w1 AND ("RotAbsPosDeg" > #HomePosAbsDeg);
   #HomeRevTorqLim_TON(IN := #_w3 AND ("ActTorqFtLbsFilt" >= "HMI_DB".OscTorqRevLowLimFtlbs),   // TON
                       PT := "Settings".OscTorqLimTime);
   IF #HomeRevTorqLim_TON.Q THEN #HomeRevTorqLim := TRUE; END_IF;
   IF #_w3 AND ("ActTorqFtLbsFilt" >= "HMI_DB".OscTorqRevHighLimFtLbs) THEN #HomeRevTorqLim := TRUE; END_IF;
   #_w4 := #_w3 AND #HomeRevTorqLim;
   #_w5 := #_w4 AND NOT #HomeRevTorqLimTrig;   // rising edge
   #HomeRevTorqLimTrig := #_w4;
   IF #_w5 THEN #LimitFlowmA := #CalcFlowmA; END_IF;
   IF #_w3 AND ("ActTorqFtLbsFilt" < "HMI_DB".OscTorqRevLowLimFtlbs) AND (#CalcFlowmA < #LimitFlowmA) THEN
       #HomeRevTorqLim := FALSE;
   END_IF;
   #_w6 := #_w3 AND #HomeRevTorqLim;
   IF #_w6 AND ("ActTorqFtLbsFilt" >= "HMI_DB".OscTorqRevHighLimFtLbs) THEN
       #HomeRevTorqLim_SlewDec(SlewRate := "HMI_DB".OscSlewFallSlow, RealValue := #LimitFlowmA);   // "SlewDec"
   END_IF;
   IF #_w6 AND ("ActTorqFtLbsFilt" < "HMI_DB".OscTorqRevLowLimFtlbs) AND "AlwaysOff" THEN
       #HomeRevTorqLim_SlewInc(SlewRate := "HMI_DB".OscSlewRiseSlow, RealValue := #LimitFlowmA);   // "SlewInc"
   END_IF;
   IF #_w6 AND NOT #PumpToggle THEN
       #CalcFlowmA := LIMIT(MN := "HMI_DB".OscP1RevMinmA, IN := #CalcFlowmA, MX := #LimitFlowmA);
       #FlowmAOut := LIMIT(MN := "HMI_DB".OscP1RevMinmA, IN := #CalcFlowmA, MX := "HMI_DB".OscP1RevMaxmA);
   END_IF;
   IF #_w6 AND #PumpToggle THEN
       #CalcFlowmA := LIMIT(MN := "HMI_DB".OscP2RevMinmA, IN := #CalcFlowmA, MX := #LimitFlowmA);
       #FlowmAOut := LIMIT(MN := "HMI_DB".OscP2RevMinmA, IN := #CalcFlowmA, MX := "HMI_DB".OscP2RevMaxmA);
   END_IF;
   #_w7 := #_w3 AND NOT #HomeRevTorqLim AND #FlowRev;
   IF #_w7 THEN #HomeDegDiff := "RotAbsPosDeg" - #HomePosAbsDeg; END_IF;
   IF #_w7 AND (#HomeDegDiff > 360.0) THEN #CalcFlowmA := "HMI_DB".OscP1RevMinmA + 150.0; END_IF;
   IF #_w7 AND (#HomeDegDiff > 180.0) AND (#HomeDegDiff < 360.0) THEN
       #CalcFlowmA := "HMI_DB".OscP1RevMinmA + 75.0;
   END_IF;
   IF #_w7 AND (#HomeDegDiff < 180.0) THEN #CalcFlowmA := "HMI_DB".OscP1RevMinmA + 55.0; END_IF;
   IF #_w7 AND NOT #PumpToggle THEN
       #FlowmAOut := LIMIT(MN := "HMI_DB".OscP1RevMinmA, IN := #CalcFlowmA, MX := "HMI_DB".OscP1RevMaxmA);
   END_IF;
   IF #_w7 AND #PumpToggle THEN
       #CalcFlowmA := #CalcFlowmA + 55.0;
       #FlowmAOut := LIMIT(MN := "HMI_DB".OscP2RevMinmA, IN := #CalcFlowmA, MX := "HMI_DB".OscP2RevMaxmA);
   END_IF;
   #_w8 := #_w1 AND ("RotAbsPosDeg" <= #HomePosAbsDeg);
   IF #_w8 THEN #OscState := #AwaitCmd; END_IF;
   IF #_w8 AND NOT #PumpToggle THEN #FlowmAOut := "HMI_DB".OscP1RevMinmA; END_IF;
   IF #_w8 AND #PumpToggle THEN #FlowmAOut := "HMI_DB".OscP2RevMinmA; END_IF;
   IF #_w8 THEN #Oscillating := FALSE; END_IF;
   IF #OscState <> #HomeRev THEN #OscRevTorqLim := FALSE; END_IF;
END_REGION

REGION Network 19: Torq Control Outputs
   // Torq is set based on Fwd torq setpoint and is enabled if not Stopped.
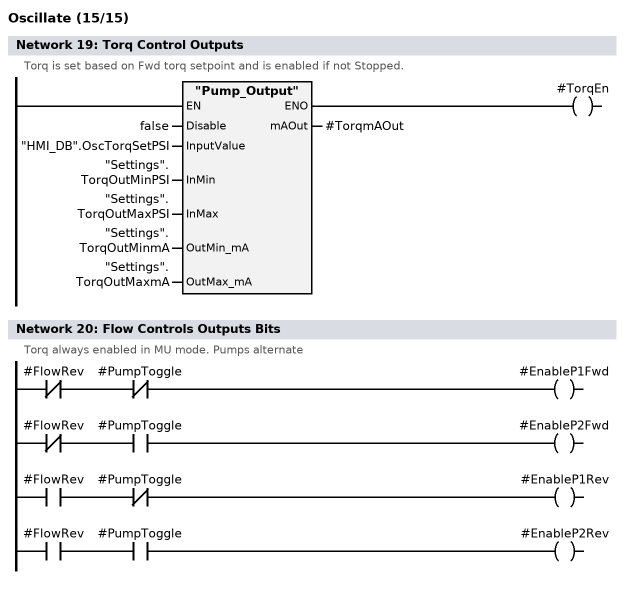
   RUNG wire#powerrail
      "Pump_Output"(Disable := false, InputValue := "HMI_DB".OscTorqSetPSI, InMin := "Settings".TorqOutMinPSI, InMax := "Settings".TorqOutMaxPSI, OutMin_mA := "Settings".TorqOutMinmA, OutMax_mA := "Settings".TorqOutMaxmA, mAOut => #TorqmAOut)
      Coil( #TorqEn )
   END_RUNG
   // the same network as SCL:
   "Pump_Output"(Disable := false,
                 InputValue := "HMI_DB".OscTorqSetPSI,
                 InMin := "Settings".TorqOutMinPSI,
                 InMax := "Settings".TorqOutMaxPSI,
                 OutMin_mA := "Settings".TorqOutMinmA,
                 OutMax_mA := "Settings".TorqOutMaxmA,
                 mAOut => #TorqmAOut,
                 ENO => #_w1);
   #TorqEn := #_w1;
END_REGION

REGION Network 20: Flow Controls Outputs Bits
   // Torq always enabled in MU mode. Pumps alternate
   RUNG wire#powerrail
      I_Contact( #FlowRev )
      I_Contact( #PumpToggle )
      Coil( #EnableP1Fwd )
   END_RUNG
   RUNG wire#powerrail
      I_Contact( #FlowRev )
      Contact( #PumpToggle )
      Coil( #EnableP2Fwd )
   END_RUNG
   RUNG wire#powerrail
      Contact( #FlowRev )
      I_Contact( #PumpToggle )
      Coil( #EnableP1Rev )
   END_RUNG
   RUNG wire#powerrail
      Contact( #FlowRev )
      Contact( #PumpToggle )
      Coil( #EnableP2Rev )
   END_RUNG
   // the same network as SCL:
   #EnableP1Fwd := NOT #FlowRev AND NOT #PumpToggle;
   #EnableP2Fwd := NOT #FlowRev AND #PumpToggle;
   #EnableP1Rev := #FlowRev AND NOT #PumpToggle;
   #EnableP2Rev := #FlowRev AND #PumpToggle;
END_REGION
END_FUNCTION_BLOCK

FUNCTION_BLOCK "Alarms"   // FB18, LAD
{ S7_Optimized_Access := 'TRUE' }
// stored: AutoNumber false, MemoryReserve 100, SetENOAutomatically false
   VAR
      BypassTempAlarm_TON { S7_SetPoint := 'True'} : TON_TIME;
      TDPressTxFaul_TON { S7_SetPoint := 'True'} : TON_TIME;
      HiTemp_TON { S7_SetPoint := 'True'} : TON_TIME;
      NoFlushFlow_TON { S7_SetPoint := 'True'} : TON_TIME;
      ChargeFault_TON { S7_SetPoint := 'True'} : TON_TIME;
      HiTempRPM_TON { S7_SetPoint := 'True'} : TON_TIME;
      HornOn_TP { S7_SetPoint := 'True'} : TP_TIME;   // Time horn is on for when request come through
      HiTempAlarm_TON { S7_SetPoint := 'True'} : TON_TIME;
      FlushFault_TP { S7_SetPoint := 'True'} : TP_TIME;
      LubeFlowFault_TON { S7_SetPoint := 'True'} : TON_TIME;
      LubeFault_TP { S7_SetPoint := 'True'} : TP_TIME;
      Charge2Fault_TON { S7_SetPoint := 'True'} : TON_TIME;
      Charge1Fault_TP { S7_SetPoint := 'True'} : TP_TIME;
      Charge2Fault_TP { S7_SetPoint := 'True'} : TP_TIME;
      FilterFault_TP { S7_SetPoint := 'True'} : TP_TIME;
      AuxPumpFault_TP { S7_SetPoint := 'True'} : TP_TIME;
      FanFault_TP { S7_SetPoint := 'True'} : TP_TIME;
      M1Fault_TP { S7_SetPoint := 'True'} : TP_TIME;
      M2Fault_TP { S7_SetPoint := 'True'} : TP_TIME;
      HiTempFault_TP { S7_SetPoint := 'True'} : TP_TIME;
      TankLevelFault_TP { S7_SetPoint := 'True'} : TP_TIME;
      TankTempFault_TP { S7_SetPoint := 'True'} : TP_TIME;
      HiTempShtdwn_TP { S7_SetPoint := 'True'} : TP_TIME;
      TDPressTXFault_TP { S7_SetPoint := 'True'} : TP_TIME;
      EngineFault_TP { S7_SetPoint := 'True'} : TP_TIME;
      BypassHiTemp_Tp { S7_SetPoint := 'True'} : TP_TIME;
      ComFault_Tp { S7_SetPoint := 'True'} : TP_TIME;
      SystemFault_Tp { S7_SetPoint := 'True'} : TP_TIME;
   END_VAR
   VAR_TEMP
      tempReal : Real;
      tempBool : Bool;
      tempTime : Time;
   END_VAR
   VAR_TEMP   // added for the SCL form of the ladder/FBD networks
      _w1 : Bool;
      _w2 : Bool;
   END_VAR
BEGIN

REGION Network 1: TD Flush Fault
   // If Aux Pump running and not in Hand and no flush within in set time disable spin
   // Aux Pump in Hand is Bypass for no flush interlock
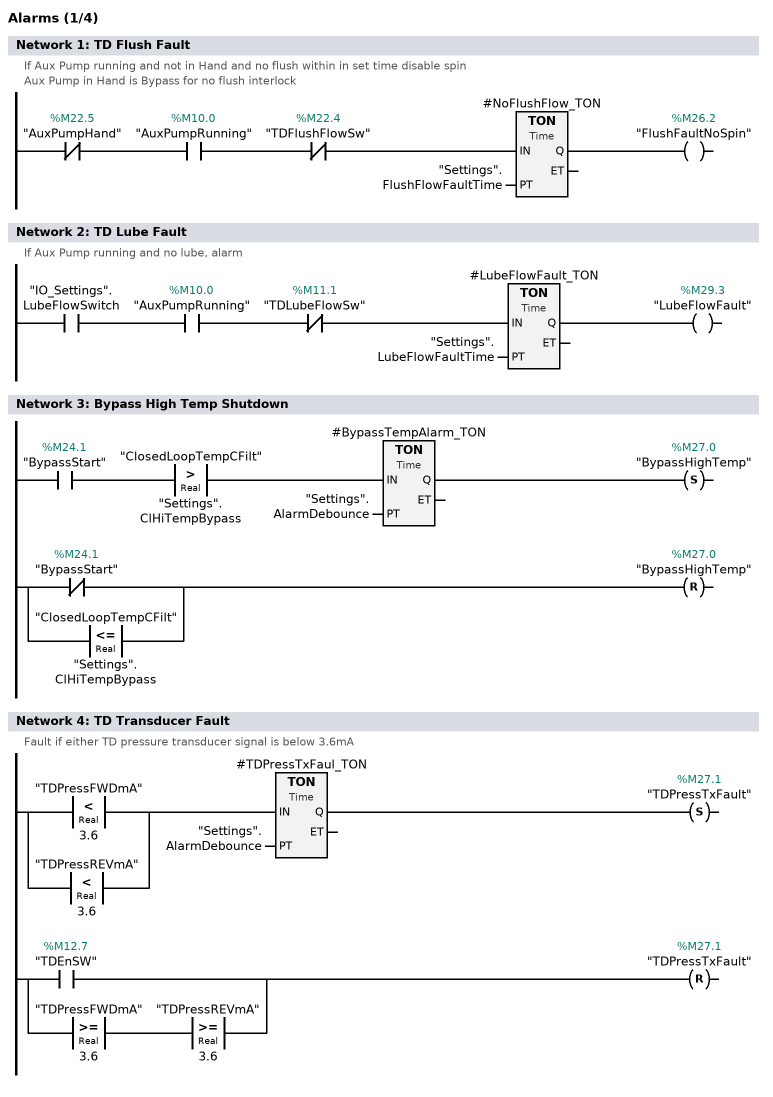
   RUNG wire#powerrail
      I_Contact( "AuxPumpHand" )
      Contact( "AuxPumpRunning" )
      I_Contact( "TDFlushFlowSw" )
      { S7_Templates := "time_type := Time" } #NoFlushFlow_TON.TON(pt := "Settings".FlushFlowFaultTime, et =>)
      Coil( "FlushFaultNoSpin" )
   END_RUNG
   // the same network as SCL:
   #NoFlushFlow_TON(IN := NOT "AuxPumpHand" AND "AuxPumpRunning" AND NOT "TDFlushFlowSw",   // TON
                    PT := "Settings".FlushFlowFaultTime);
   "FlushFaultNoSpin" := #NoFlushFlow_TON.Q;
END_REGION

REGION Network 2: TD Lube Fault
   // If Aux Pump running and no lube, alarm
   RUNG wire#powerrail
      Contact( "IO_Settings".LubeFlowSwitch )
      Contact( "AuxPumpRunning" )
      I_Contact( "TDLubeFlowSw" )
      { S7_Templates := "time_type := Time" } #LubeFlowFault_TON.TON(pt := "Settings".LubeFlowFaultTime, et =>)
      Coil( "LubeFlowFault" )
   END_RUNG
   // the same network as SCL:
   #LubeFlowFault_TON(IN := "IO_Settings".LubeFlowSwitch AND "AuxPumpRunning" AND NOT "TDLubeFlowSw",   // TON
                      PT := "Settings".LubeFlowFaultTime);
   "LubeFlowFault" := #LubeFlowFault_TON.Q;
END_REGION

REGION Network 3: Bypass High Temp Shutdown
   RUNG wire#powerrail
      Contact( "BypassStart" )
      { S7_Templates := "SrcType := Real" } GT_Contact(in1 := "ClosedLoopTempCFilt", in2 := "Settings".ClHiTempBypass)
      { S7_Templates := "time_type := Time" } #BypassTempAlarm_TON.TON(pt := "Settings".AlarmDebounce, et =>)
      S_Coil( "BypassHighTemp" )
   END_RUNG
   RUNG wire#powerrail
      I_Contact( "BypassStart" )
      wire#w1
      R_Coil( "BypassHighTemp" )
   END_RUNG
   RUNG wire#powerrail
      { S7_Templates := "SrcType := Real" } LE_Contact(in1 := "ClosedLoopTempCFilt", in2 := "Settings".ClHiTempBypass)
   END_RUNG wire#w1
   // the same network as SCL:
   #BypassTempAlarm_TON(IN := "BypassStart" AND ("ClosedLoopTempCFilt" > "Settings".ClHiTempBypass),   // TON
                        PT := "Settings".AlarmDebounce);
   IF #BypassTempAlarm_TON.Q THEN "BypassHighTemp" := TRUE; END_IF;
   IF NOT "BypassStart" OR ("ClosedLoopTempCFilt" <= "Settings".ClHiTempBypass) THEN
       "BypassHighTemp" := FALSE;
   END_IF;
END_REGION

REGION Network 4: TD Transducer Fault
   // Fault if either TD pressure transducer signal is below 3.6mA
   RUNG wire#powerrail
      { S7_Templates := "SrcType := Real" } LT_Contact(in1 := "TDPressFWDmA", in2 := 3.6)
      wire#w1
      { S7_Templates := "time_type := Time" } #TDPressTxFaul_TON.TON(pt := "Settings".AlarmDebounce, et =>)
      S_Coil( "TDPressTxFault" )
   END_RUNG
   RUNG wire#powerrail
      { S7_Templates := "SrcType := Real" } LT_Contact(in1 := "TDPressREVmA", in2 := 3.6)
   END_RUNG wire#w1
   RUNG wire#powerrail
      Contact( "TDEnSW" )
      wire#w2
      R_Coil( "TDPressTxFault" )
   END_RUNG
   RUNG wire#powerrail
      { S7_Templates := "SrcType := Real" } GE_Contact(in1 := "TDPressFWDmA", in2 := 3.6)
      { S7_Templates := "SrcType := Real" } GE_Contact(in1 := "TDPressREVmA", in2 := 3.6)
   END_RUNG wire#w2
   // the same network as SCL:
   #TDPressTxFaul_TON(IN := ("TDPressFWDmA" < 3.6) OR ("TDPressREVmA" < 3.6), PT := "Settings".AlarmDebounce);   // TON
   IF #TDPressTxFaul_TON.Q THEN "TDPressTxFault" := TRUE; END_IF;
   IF "TDEnSW" OR (("TDPressFWDmA" >= 3.6) AND ("TDPressREVmA" >= 3.6)) THEN
       "TDPressTxFault" := FALSE;
   END_IF;
END_REGION

REGION Network 5: Closed Loop High Temp Shutdown
   // Reduce RPM if temp above RPM reduction temp
   // Shudown if temp above shutdown.
   // Reset either when 3 C below trigger point
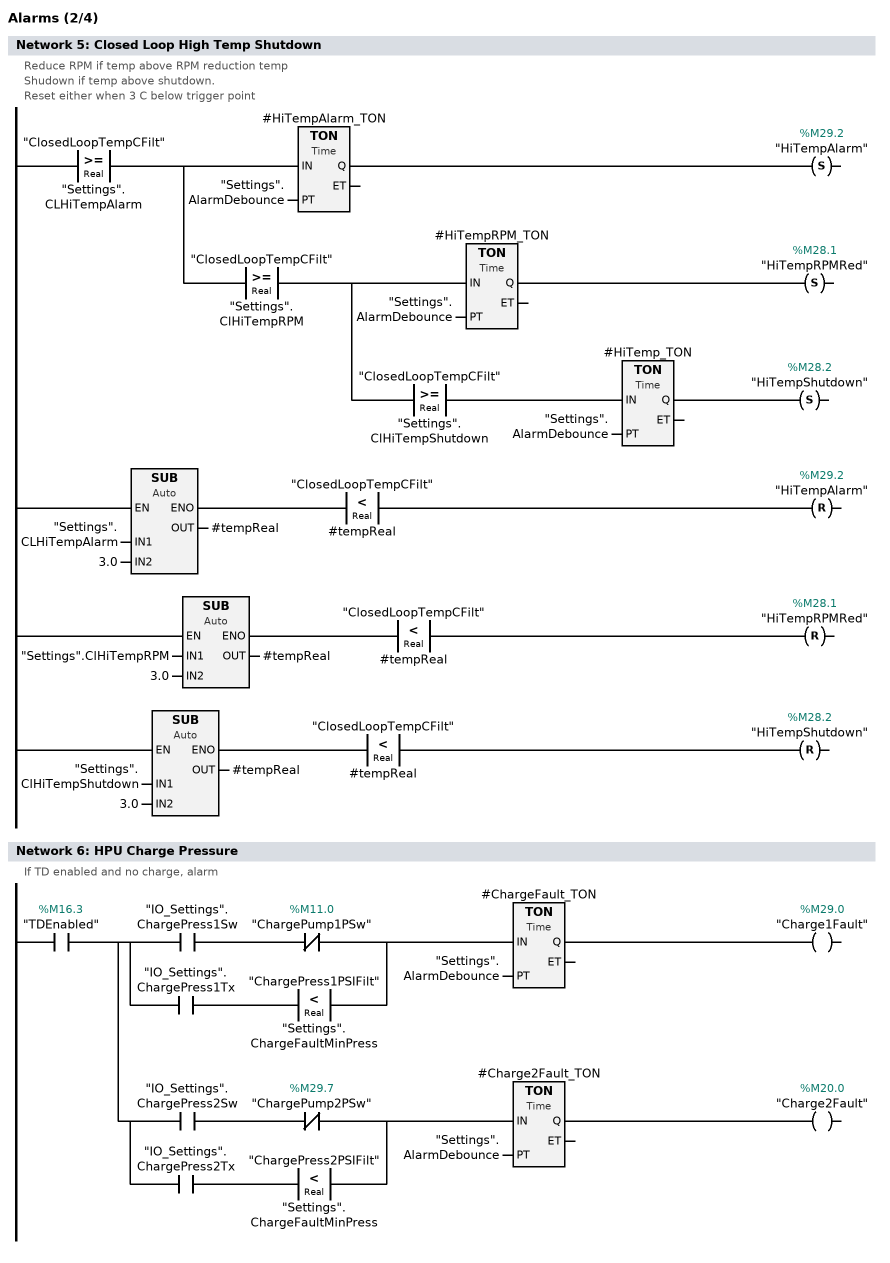
   RUNG wire#powerrail
      { S7_Templates := "SrcType := Real" } GE_Contact(in1 := "ClosedLoopTempCFilt", in2 := "Settings".CLHiTempAlarm)
      wire#w1
      { S7_Templates := "time_type := Time" } #HiTempAlarm_TON.TON(pt := "Settings".AlarmDebounce, et =>)
      S_Coil( "HiTempAlarm" )
   END_RUNG
   RUNG wire#w1
      { S7_Templates := "SrcType := Real" } GE_Contact(in1 := "ClosedLoopTempCFilt", in2 := "Settings".ClHiTempRPM)
      wire#w2
      { S7_Templates := "time_type := Time" } #HiTempRPM_TON.TON(pt := "Settings".AlarmDebounce, et =>)
      S_Coil( "HiTempRPMRed" )
   END_RUNG
   RUNG wire#w2
      { S7_Templates := "SrcType := Real" } GE_Contact(in1 := "ClosedLoopTempCFilt", in2 := "Settings".ClHiTempShutdown)
      { S7_Templates := "time_type := Time" } #HiTemp_TON.TON(pt := "Settings".AlarmDebounce, et =>)
      S_Coil( "HiTempShutdown" )
   END_RUNG
   RUNG wire#powerrail
      Sub(in1 := "Settings".CLHiTempAlarm, in2 := 3.0, out => #tempReal)
      { S7_Templates := "SrcType := Real" } LT_Contact(in1 := "ClosedLoopTempCFilt", in2 := #tempReal)
      R_Coil( "HiTempAlarm" )
   END_RUNG
   RUNG wire#powerrail
      Sub(in1 := "Settings".ClHiTempRPM, in2 := 3.0, out => #tempReal)
      { S7_Templates := "SrcType := Real" } LT_Contact(in1 := "ClosedLoopTempCFilt", in2 := #tempReal)
      R_Coil( "HiTempRPMRed" )
   END_RUNG
   RUNG wire#powerrail
      Sub(in1 := "Settings".ClHiTempShutdown, in2 := 3.0, out => #tempReal)
      { S7_Templates := "SrcType := Real" } LT_Contact(in1 := "ClosedLoopTempCFilt", in2 := #tempReal)
      R_Coil( "HiTempShutdown" )
   END_RUNG
   // the same network as SCL:
   #_w1 := "ClosedLoopTempCFilt" >= "Settings".CLHiTempAlarm;
   #HiTempAlarm_TON(IN := #_w1, PT := "Settings".AlarmDebounce);   // TON
   IF #HiTempAlarm_TON.Q THEN "HiTempAlarm" := TRUE; END_IF;
   #_w2 := #_w1 AND ("ClosedLoopTempCFilt" >= "Settings".ClHiTempRPM);
   #HiTempRPM_TON(IN := #_w2, PT := "Settings".AlarmDebounce);   // TON
   IF #HiTempRPM_TON.Q THEN "HiTempRPMRed" := TRUE; END_IF;
   #HiTemp_TON(IN := #_w2 AND ("ClosedLoopTempCFilt" >= "Settings".ClHiTempShutdown),   // TON
               PT := "Settings".AlarmDebounce);
   IF #HiTemp_TON.Q THEN "HiTempShutdown" := TRUE; END_IF;
   #tempReal := "Settings".CLHiTempAlarm - 3.0;
   IF "ClosedLoopTempCFilt" < #tempReal THEN "HiTempAlarm" := FALSE; END_IF;
   #tempReal := "Settings".ClHiTempRPM - 3.0;
   IF "ClosedLoopTempCFilt" < #tempReal THEN "HiTempRPMRed" := FALSE; END_IF;
   #tempReal := "Settings".ClHiTempShutdown - 3.0;
   IF "ClosedLoopTempCFilt" < #tempReal THEN "HiTempShutdown" := FALSE; END_IF;
END_REGION

REGION Network 6: HPU Charge Pressure
   // If TD enabled and no charge, alarm
   RUNG wire#powerrail
      Contact( "TDEnabled" )
      wire#w1
      Contact( "IO_Settings".ChargePress1Sw )
      I_Contact( "ChargePump1PSw" )
      wire#w2
      { S7_Templates := "time_type := Time" } #ChargeFault_TON.TON(pt := "Settings".AlarmDebounce, et =>)
      Coil( "Charge1Fault" )
   END_RUNG
   RUNG wire#w1
      Contact( "IO_Settings".ChargePress1Tx )
      { S7_Templates := "SrcType := Real" } LT_Contact(in1 := "ChargePress1PSIFilt", in2 := "Settings".ChargeFaultMinPress)
   END_RUNG wire#w2
   RUNG wire#w1
      Contact( "IO_Settings".ChargePress2Sw )
      I_Contact( "ChargePump2PSw" )
      wire#w3
      { S7_Templates := "time_type := Time" } #Charge2Fault_TON.TON(pt := "Settings".AlarmDebounce, et =>)
      Coil( "Charge2Fault" )
   END_RUNG
   RUNG wire#w1
      Contact( "IO_Settings".ChargePress2Tx )
      { S7_Templates := "SrcType := Real" } LT_Contact(in1 := "ChargePress2PSIFilt", in2 := "Settings".ChargeFaultMinPress)
   END_RUNG wire#w3
   // the same network as SCL:
   #ChargeFault_TON(IN := "TDEnabled" AND (("IO_Settings".ChargePress1Sw AND NOT "ChargePump1PSw") OR ("IO_Settings".ChargePress1Tx AND ("ChargePress1PSIFilt" < "Settings".ChargeFaultMinPress))),   // TON
                    PT := "Settings".AlarmDebounce);
   "Charge1Fault" := #ChargeFault_TON.Q;
   #Charge2Fault_TON(IN := "TDEnabled" AND (("IO_Settings".ChargePress2Sw AND NOT "ChargePump2PSw") OR ("IO_Settings".ChargePress2Tx AND ("ChargePress2PSIFilt" < "Settings".ChargeFaultMinPress))),   // TON
                     PT := "Settings".AlarmDebounce);
   "Charge2Fault" := #Charge2Fault_TON.Q;
END_REGION

REGION Network 7: Plug Filter
   // Set if any filter is plugged or charge above 1000
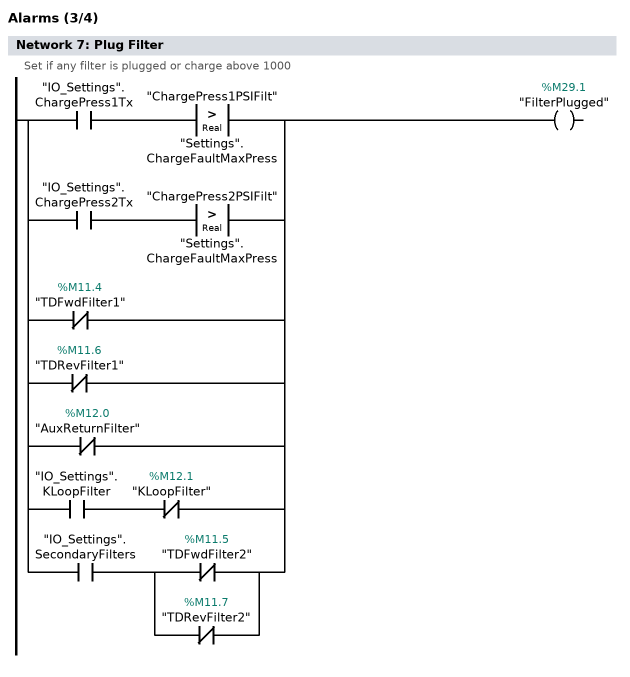
   RUNG wire#powerrail
      Contact( "IO_Settings".ChargePress1Tx )
      { S7_Templates := "SrcType := Real" } GT_Contact(in1 := "ChargePress1PSIFilt", in2 := "Settings".ChargeFaultMaxPress)
      wire#w1
      Coil( "FilterPlugged" )
   END_RUNG
   RUNG wire#powerrail
      Contact( "IO_Settings".ChargePress2Tx )
      { S7_Templates := "SrcType := Real" } GT_Contact(in1 := "ChargePress2PSIFilt", in2 := "Settings".ChargeFaultMaxPress)
   END_RUNG wire#w1
   RUNG wire#powerrail
      I_Contact( "TDFwdFilter1" )
   END_RUNG wire#w1
   RUNG wire#powerrail
      I_Contact( "TDRevFilter1" )
   END_RUNG wire#w1
   RUNG wire#powerrail
      I_Contact( "AuxReturnFilter" )
   END_RUNG wire#w1
   RUNG wire#powerrail
      Contact( "IO_Settings".KLoopFilter )
      I_Contact( "KLoopFilter" )
   END_RUNG wire#w1
   RUNG wire#powerrail
      Contact( "IO_Settings".SecondaryFilters )
      wire#w2
      I_Contact( "TDFwdFilter2" )
   END_RUNG wire#w1
   RUNG wire#w2
      I_Contact( "TDRevFilter2" )
   END_RUNG wire#w1
   // the same network as SCL:
   "FilterPlugged" := ("IO_Settings".ChargePress1Tx AND ("ChargePress1PSIFilt" > "Settings".ChargeFaultMaxPress)) OR ("IO_Settings".ChargePress2Tx AND ("ChargePress2PSIFilt" > "Settings".ChargeFaultMaxPress)) OR NOT "TDFwdFilter1" OR NOT "TDRevFilter1" OR NOT "AuxReturnFilter" OR ("IO_Settings".KLoopFilter AND NOT "KLoopFilter") OR ("IO_Settings".SecondaryFilters AND (NOT "TDFwdFilter2" OR NOT "TDRevFilter2"));
END_REGION

REGION Network 8: Horn
   // Turn on Horn if test or
   // Sequence Pulse for horn time if any of following faults have a pulsed:
   // FlushFault/Low Level/Tank Temp/LubeFault/FilterPlugged/Any Motor Start Fault/Charge Pressure fault, engine fault.
   // Clock Horn for High Temp unless silenced
   // Trigger horn 1 a minute if reduced RPM.
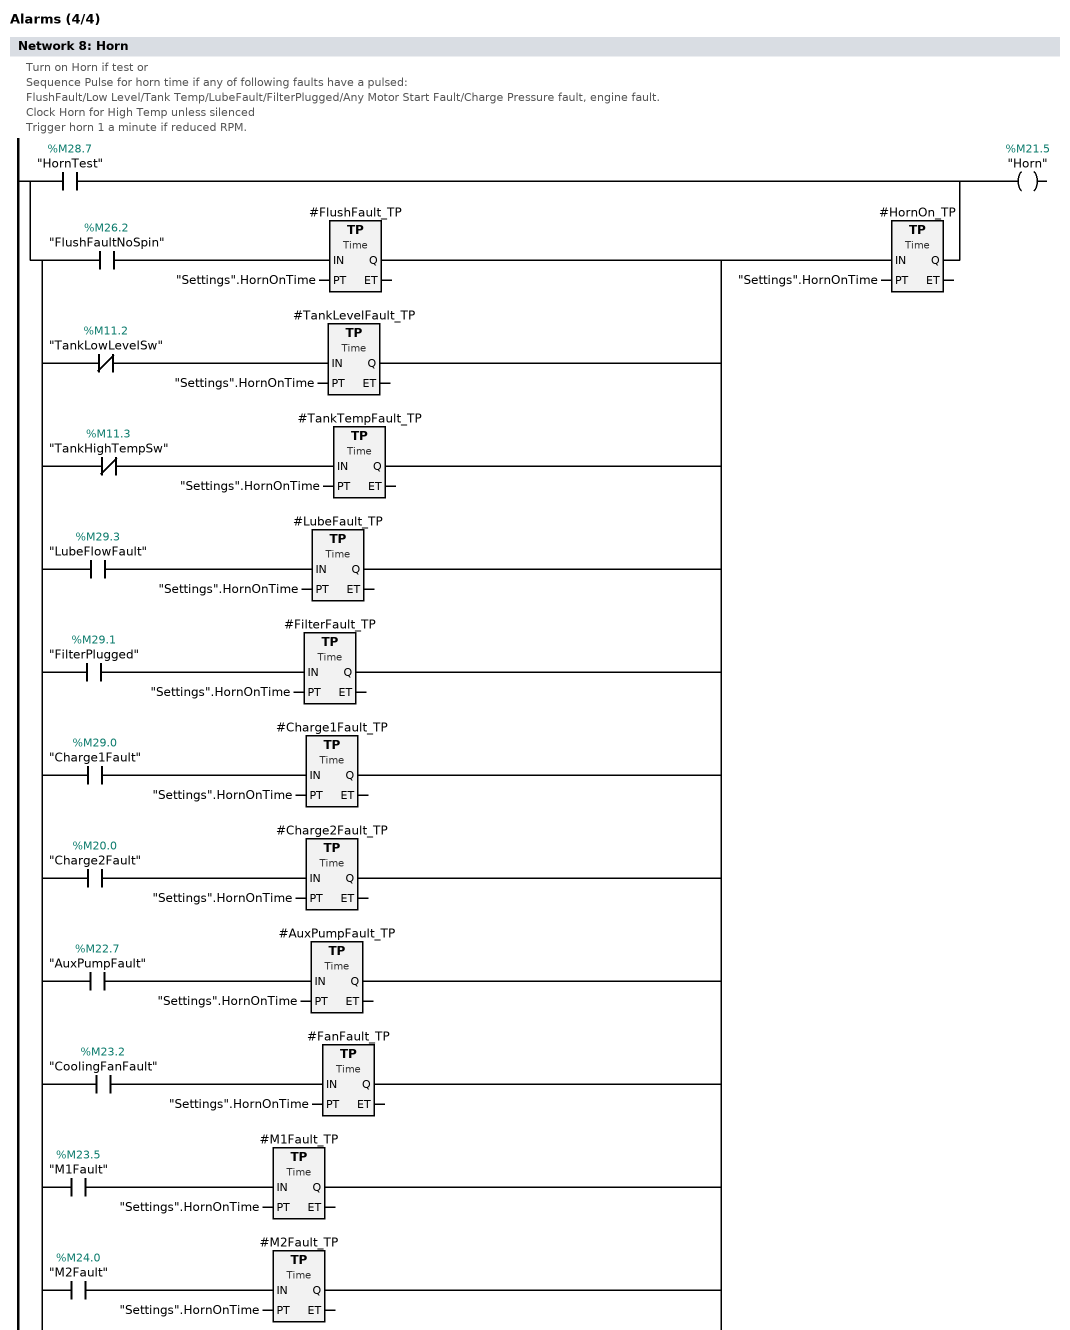
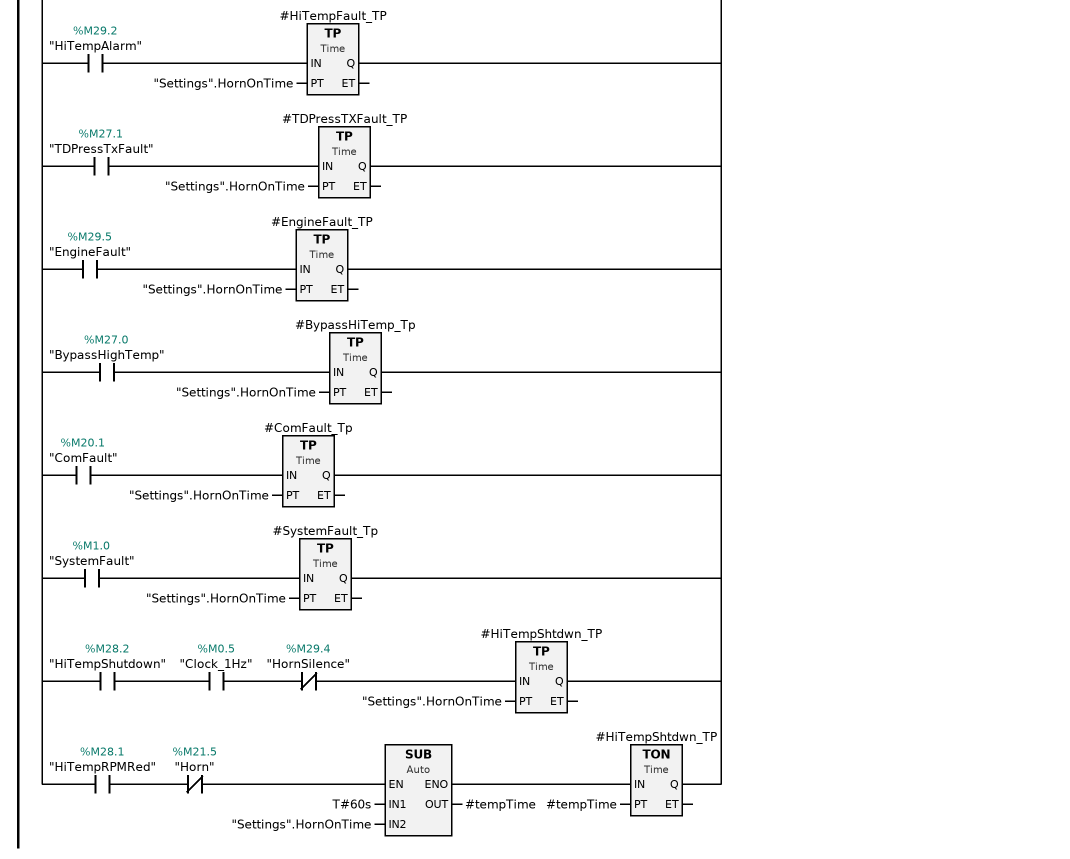
   RUNG wire#powerrail
      Contact( "HornTest" )
      wire#w1
      Coil( "Horn" )
   END_RUNG
   RUNG wire#powerrail
      Contact( "FlushFaultNoSpin" )
      { S7_Templates := "time_type := Time" } #FlushFault_TP.TP(pt := "Settings".HornOnTime, et =>)
      wire#w2
      { S7_Templates := "time_type := Time" } #HornOn_TP.TP(pt := "Settings".HornOnTime, et =>)
   END_RUNG wire#w1
   RUNG wire#powerrail
      I_Contact( "TankLowLevelSw" )
      { S7_Templates := "time_type := Time" } #TankLevelFault_TP.TP(pt := "Settings".HornOnTime, et =>)
   END_RUNG wire#w2
   RUNG wire#powerrail
      I_Contact( "TankHighTempSw" )
      { S7_Templates := "time_type := Time" } #TankTempFault_TP.TP(pt := "Settings".HornOnTime, et =>)
   END_RUNG wire#w2
   RUNG wire#powerrail
      Contact( "LubeFlowFault" )
      { S7_Templates := "time_type := Time" } #LubeFault_TP.TP(pt := "Settings".HornOnTime, et =>)
   END_RUNG wire#w2
   RUNG wire#powerrail
      Contact( "FilterPlugged" )
      { S7_Templates := "time_type := Time" } #FilterFault_TP.TP(pt := "Settings".HornOnTime, et =>)
   END_RUNG wire#w2
   RUNG wire#powerrail
      Contact( "Charge1Fault" )
      { S7_Templates := "time_type := Time" } #Charge1Fault_TP.TP(pt := "Settings".HornOnTime, et =>)
   END_RUNG wire#w2
   RUNG wire#powerrail
      Contact( "Charge2Fault" )
      { S7_Templates := "time_type := Time" } #Charge2Fault_TP.TP(pt := "Settings".HornOnTime, et =>)
   END_RUNG wire#w2
   RUNG wire#powerrail
      Contact( "AuxPumpFault" )
      { S7_Templates := "time_type := Time" } #AuxPumpFault_TP.TP(pt := "Settings".HornOnTime, et =>)
   END_RUNG wire#w2
   RUNG wire#powerrail
      Contact( "CoolingFanFault" )
      { S7_Templates := "time_type := Time" } #FanFault_TP.TP(pt := "Settings".HornOnTime, et =>)
   END_RUNG wire#w2
   RUNG wire#powerrail
      Contact( "M1Fault" )
      { S7_Templates := "time_type := Time" } #M1Fault_TP.TP(pt := "Settings".HornOnTime, et =>)
   END_RUNG wire#w2
   RUNG wire#powerrail
      Contact( "M2Fault" )
      { S7_Templates := "time_type := Time" } #M2Fault_TP.TP(pt := "Settings".HornOnTime, et =>)
   END_RUNG wire#w2
   RUNG wire#powerrail
      Contact( "HiTempAlarm" )
      { S7_Templates := "time_type := Time" } #HiTempFault_TP.TP(pt := "Settings".HornOnTime, et =>)
   END_RUNG wire#w2
   RUNG wire#powerrail
      Contact( "TDPressTxFault" )
      { S7_Templates := "time_type := Time" } #TDPressTXFault_TP.TP(pt := "Settings".HornOnTime, et =>)
   END_RUNG wire#w2
   RUNG wire#powerrail
      Contact( "EngineFault" )
      { S7_Templates := "time_type := Time" } #EngineFault_TP.TP(pt := "Settings".HornOnTime, et =>)
   END_RUNG wire#w2
   RUNG wire#powerrail
      Contact( "BypassHighTemp" )
      { S7_Templates := "time_type := Time" } #BypassHiTemp_Tp.TP(pt := "Settings".HornOnTime, et =>)
   END_RUNG wire#w2
   RUNG wire#powerrail
      Contact( "ComFault" )
      { S7_Templates := "time_type := Time" } #ComFault_Tp.TP(pt := "Settings".HornOnTime, et =>)
   END_RUNG wire#w2
   RUNG wire#powerrail
      Contact( "SystemFault" )
      { S7_Templates := "time_type := Time" } #SystemFault_Tp.TP(pt := "Settings".HornOnTime, et =>)
   END_RUNG wire#w2
   RUNG wire#powerrail
      Contact( "HiTempShutdown" )
      Contact( "Clock_1Hz" )
      I_Contact( "HornSilence" )
      { S7_Templates := "time_type := Time" } #HiTempShtdwn_TP.TP(pt := "Settings".HornOnTime, et =>)
   END_RUNG wire#w2
   RUNG wire#powerrail
      Contact( "HiTempRPMRed" )
      I_Contact( "Horn" )
      Sub(in1 := T#60s, in2 := "Settings".HornOnTime, out => #tempTime)
      { S7_Templates := "time_type := Time" } #HiTempShtdwn_TP.TON(pt := #tempTime, et =>)
   END_RUNG wire#w2
   // the same network as SCL:
   #FlushFault_TP(IN := "FlushFaultNoSpin", PT := "Settings".HornOnTime);   // TP
   #TankLevelFault_TP(IN := NOT "TankLowLevelSw", PT := "Settings".HornOnTime);   // TP
   #TankTempFault_TP(IN := NOT "TankHighTempSw", PT := "Settings".HornOnTime);   // TP
   #LubeFault_TP(IN := "LubeFlowFault", PT := "Settings".HornOnTime);   // TP
   #FilterFault_TP(IN := "FilterPlugged", PT := "Settings".HornOnTime);   // TP
   #Charge1Fault_TP(IN := "Charge1Fault", PT := "Settings".HornOnTime);   // TP
   #Charge2Fault_TP(IN := "Charge2Fault", PT := "Settings".HornOnTime);   // TP
   #AuxPumpFault_TP(IN := "AuxPumpFault", PT := "Settings".HornOnTime);   // TP
   #FanFault_TP(IN := "CoolingFanFault", PT := "Settings".HornOnTime);   // TP
   #M1Fault_TP(IN := "M1Fault", PT := "Settings".HornOnTime);   // TP
   #M2Fault_TP(IN := "M2Fault", PT := "Settings".HornOnTime);   // TP
   #HiTempFault_TP(IN := "HiTempAlarm", PT := "Settings".HornOnTime);   // TP
   #TDPressTXFault_TP(IN := "TDPressTxFault", PT := "Settings".HornOnTime);   // TP
   #EngineFault_TP(IN := "EngineFault", PT := "Settings".HornOnTime);   // TP
   #BypassHiTemp_Tp(IN := "BypassHighTemp", PT := "Settings".HornOnTime);   // TP
   #ComFault_Tp(IN := "ComFault", PT := "Settings".HornOnTime);   // TP
   #SystemFault_Tp(IN := "SystemFault", PT := "Settings".HornOnTime);   // TP
   #HiTempShtdwn_TP(IN := "HiTempShutdown" AND "Clock_1Hz" AND NOT "HornSilence", PT := "Settings".HornOnTime);   // TP
   #_w1 := "HiTempRPMRed" AND NOT "Horn";
   IF #_w1 THEN #tempTime := T#60s - "Settings".HornOnTime; END_IF;
   #_w2 := #HiTempShtdwn_TP.Q;
   #HiTempShtdwn_TP(IN := #_w1, PT := #tempTime);   // TON
   #HornOn_TP(IN := #FlushFault_TP.Q OR #TankLevelFault_TP.Q OR #TankTempFault_TP.Q OR #LubeFault_TP.Q OR #FilterFault_TP.Q OR #Charge1Fault_TP.Q OR #Charge2Fault_TP.Q OR #AuxPumpFault_TP.Q OR #FanFault_TP.Q OR #M1Fault_TP.Q OR #M2Fault_TP.Q OR #HiTempFault_TP.Q OR #TDPressTXFault_TP.Q OR #EngineFault_TP.Q OR #BypassHiTemp_Tp.Q OR #ComFault_Tp.Q OR #SystemFault_Tp.Q OR #_w2 OR #HiTempShtdwn_TP.Q,   // TP
              PT := "Settings".HornOnTime);
   "Horn" := "HornTest" OR #HornOn_TP.Q;
END_REGION
END_FUNCTION_BLOCK

FUNCTION_BLOCK "LEDS"   // FB17, LAD
{ S7_Optimized_Access := 'TRUE' }
// stored: AutoNumber false, MemoryReserve 100, SetENOAutomatically false
   VAR
      ElevClLEDStatus : Bool;
      MSVClLEDStatus : Bool;
      BUWClLEDStatus : Bool;
   END_VAR
   VAR_TEMP
      BUWClLEDOffDely : Bool;
   END_VAR
BEGIN

REGION Network 1: Elev Closed LED
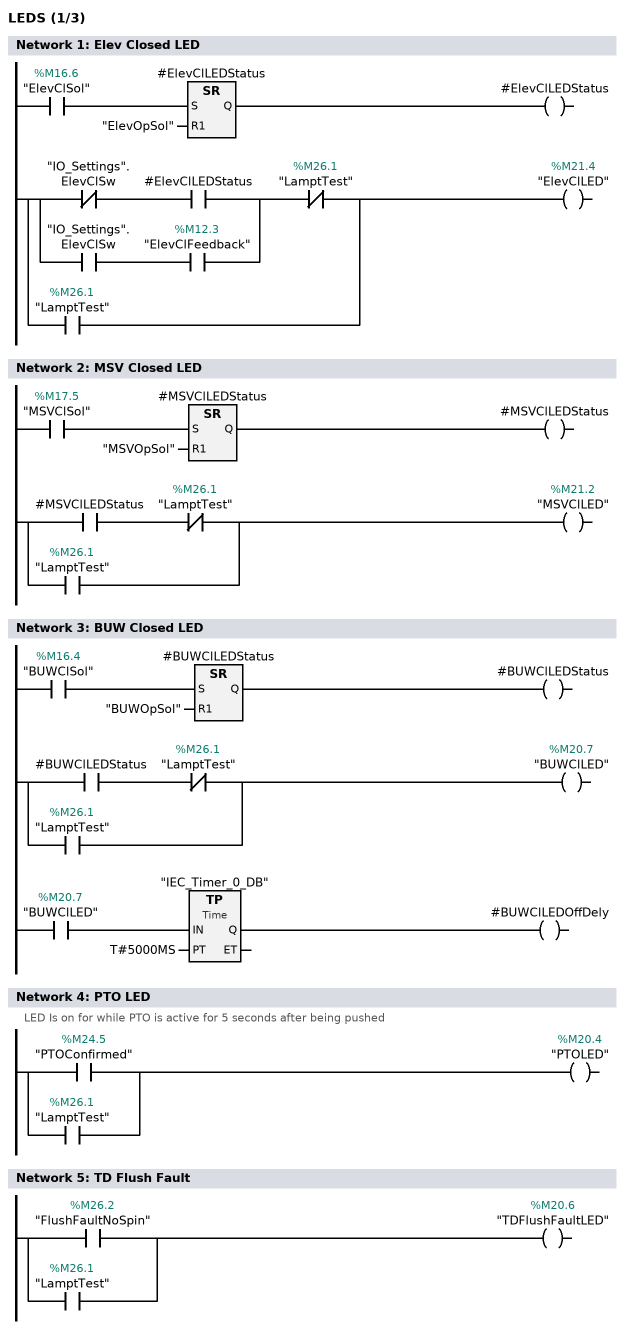
   RUNG wire#powerrail
      Contact( "ElevClSol" )
      S_SR(operand := #ElevClLEDStatus, r1 := "ElevOpSol")
      Coil( #ElevClLEDStatus )
   END_RUNG
   RUNG wire#powerrail
      I_Contact( "IO_Settings".ElevClSw )
      Contact( #ElevClLEDStatus )
      wire#w1
      I_Contact( "LamptTest" )
      wire#w2
      Coil( "ElevClLED" )
   END_RUNG
   RUNG wire#powerrail
      Contact( "IO_Settings".ElevClSw )
      Contact( "ElevClFeedback" )
   END_RUNG wire#w1
   RUNG wire#powerrail
      Contact( "LamptTest" )
   END_RUNG wire#w2
   // the same network as SCL:
   IF "ElevClSol" THEN
       #ElevClLEDStatus := TRUE;   // SR flip-flop
   END_IF;
   IF "ElevOpSol" THEN #ElevClLEDStatus := FALSE; END_IF;
   #ElevClLEDStatus := #ElevClLEDStatus;
   "ElevClLED" := (((NOT "IO_Settings".ElevClSw AND #ElevClLEDStatus) OR ("IO_Settings".ElevClSw AND "ElevClFeedback")) AND NOT "LamptTest") OR "LamptTest";
END_REGION

REGION Network 2: MSV Closed LED
   RUNG wire#powerrail
      Contact( "MSVClSol" )
      S_SR(operand := #MSVClLEDStatus, r1 := "MSVOpSol")
      Coil( #MSVClLEDStatus )
   END_RUNG
   RUNG wire#powerrail
      Contact( #MSVClLEDStatus )
      I_Contact( "LamptTest" )
      wire#w1
      Coil( "MSVClLED" )
   END_RUNG
   RUNG wire#powerrail
      Contact( "LamptTest" )
   END_RUNG wire#w1
   // the same network as SCL:
   IF "MSVClSol" THEN
       #MSVClLEDStatus := TRUE;   // SR flip-flop
   END_IF;
   IF "MSVOpSol" THEN #MSVClLEDStatus := FALSE; END_IF;
   #MSVClLEDStatus := #MSVClLEDStatus;
   "MSVClLED" := (#MSVClLEDStatus AND NOT "LamptTest") OR "LamptTest";
END_REGION

REGION Network 3: BUW Closed LED
   RUNG wire#powerrail
      Contact( "BUWClSol" )
      S_SR(operand := #BUWClLEDStatus, r1 := "BUWOpSol")
      Coil( #BUWClLEDStatus )
   END_RUNG
   RUNG wire#powerrail
      Contact( #BUWClLEDStatus )
      I_Contact( "LamptTest" )
      wire#w1
      Coil( "BUWClLED" )
   END_RUNG
   RUNG wire#powerrail
      Contact( "LamptTest" )
   END_RUNG wire#w1
   RUNG wire#powerrail
      Contact( "BUWClLED" )
      { S7_Templates := "time_type := Time" } "IEC_Timer_0_DB".TP(pt := T#5000MS, et =>)
      Coil( #BUWClLEDOffDely )
   END_RUNG
   // the same network as SCL:
   IF "BUWClSol" THEN
       #BUWClLEDStatus := TRUE;   // SR flip-flop
   END_IF;
   IF "BUWOpSol" THEN #BUWClLEDStatus := FALSE; END_IF;
   #BUWClLEDStatus := #BUWClLEDStatus;
   "BUWClLED" := (#BUWClLEDStatus AND NOT "LamptTest") OR "LamptTest";
   "IEC_Timer_0_DB".TP(IN := "BUWClLED", PT := T#5000MS);
   #BUWClLEDOffDely := "IEC_Timer_0_DB".Q;
END_REGION

REGION Network 4: PTO LED
   // LED Is on for while PTO is active for 5 seconds after being pushed
   RUNG wire#powerrail
      Contact( "PTOConfirmed" )
      wire#w1
      Coil( "PTOLED" )
   END_RUNG
   RUNG wire#powerrail
      Contact( "LamptTest" )
   END_RUNG wire#w1
   // the same network as SCL:
   "PTOLED" := "PTOConfirmed" OR "LamptTest";
END_REGION

REGION Network 5: TD Flush Fault
   RUNG wire#powerrail
      Contact( "FlushFaultNoSpin" )
      wire#w1
      Coil( "TDFlushFaultLED" )
   END_RUNG
   RUNG wire#powerrail
      Contact( "LamptTest" )
   END_RUNG wire#w1
   // the same network as SCL:
   "TDFlushFaultLED" := "FlushFaultNoSpin" OR "LamptTest";
END_REGION

REGION Network 6: Quill Lock LED
   // IF Quill Lock, Lock Maintained and BUW is closed,(LED is ON) then Quill Lock
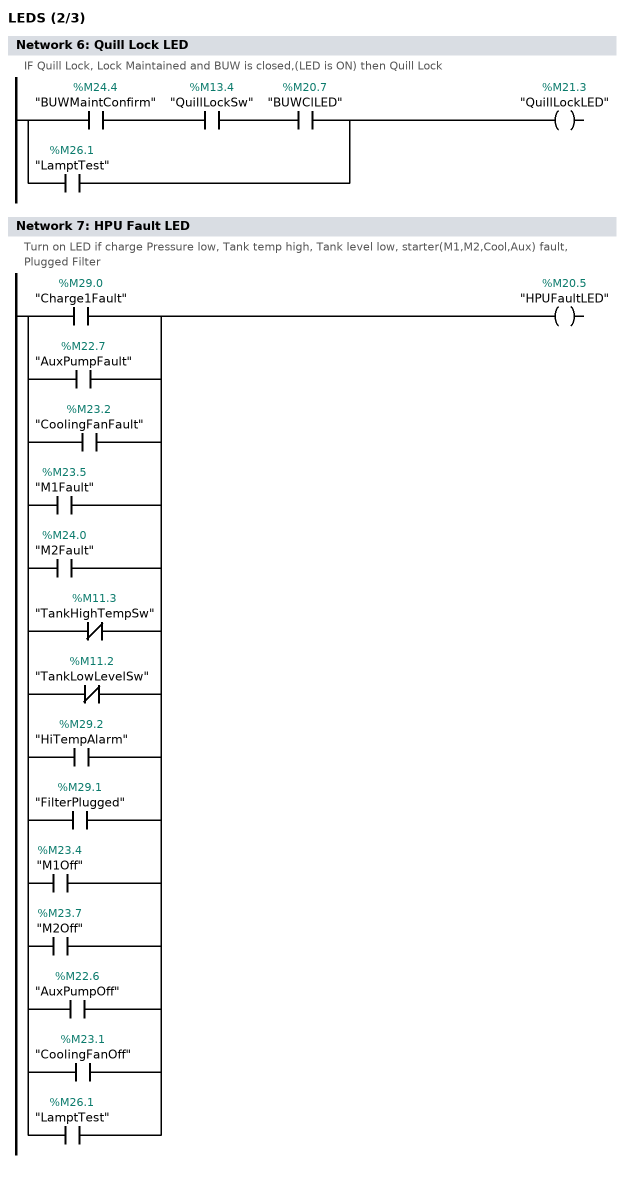
   RUNG wire#powerrail
      Contact( "BUWMaintConfirm" )
      Contact( "QuillLockSw" )
      Contact( "BUWClLED" )
      wire#w1
      Coil( "QuillLockLED" )
   END_RUNG
   RUNG wire#powerrail
      Contact( "LamptTest" )
   END_RUNG wire#w1
   // the same network as SCL:
   "QuillLockLED" := ("BUWMaintConfirm" AND "QuillLockSw" AND "BUWClLED") OR "LamptTest";
END_REGION

REGION Network 7: HPU Fault LED
   // Turn on LED if charge Pressure low, Tank temp high, Tank level low, starter(M1,M2,Cool,Aux) fault, Plugged Filter
   RUNG wire#powerrail
      Contact( "Charge1Fault" )
      wire#w1
      Coil( "HPUFaultLED" )
   END_RUNG
   RUNG wire#powerrail
      Contact( "AuxPumpFault" )
   END_RUNG wire#w1
   RUNG wire#powerrail
      Contact( "CoolingFanFault" )
   END_RUNG wire#w1
   RUNG wire#powerrail
      Contact( "M1Fault" )
   END_RUNG wire#w1
   RUNG wire#powerrail
      Contact( "M2Fault" )
   END_RUNG wire#w1
   RUNG wire#powerrail
      I_Contact( "TankHighTempSw" )
   END_RUNG wire#w1
   RUNG wire#powerrail
      I_Contact( "TankLowLevelSw" )
   END_RUNG wire#w1
   RUNG wire#powerrail
      Contact( "HiTempAlarm" )
   END_RUNG wire#w1
   RUNG wire#powerrail
      Contact( "FilterPlugged" )
   END_RUNG wire#w1
   RUNG wire#powerrail
      Contact( "M1Off" )
   END_RUNG wire#w1
   RUNG wire#powerrail
      Contact( "M2Off" )
   END_RUNG wire#w1
   RUNG wire#powerrail
      Contact( "AuxPumpOff" )
   END_RUNG wire#w1
   RUNG wire#powerrail
      Contact( "CoolingFanOff" )
   END_RUNG wire#w1
   RUNG wire#powerrail
      Contact( "LamptTest" )
   END_RUNG wire#w1
   // the same network as SCL:
   "HPUFaultLED" := "Charge1Fault" OR "AuxPumpFault" OR "CoolingFanFault" OR "M1Fault" OR "M2Fault" OR NOT "TankHighTempSw" OR NOT "TankLowLevelSw" OR "HiTempAlarm" OR "FilterPlugged" OR "M1Off" OR "M2Off" OR "AuxPumpOff" OR "CoolingFanOff" OR "LamptTest";
END_REGION

REGION Network 8: TD Enabled LED
   // If Start signal sent and enabled, Pump not in Hand and throttle not disabled than on. 
   // If Start and disabled or in hand or throttle disabled blink
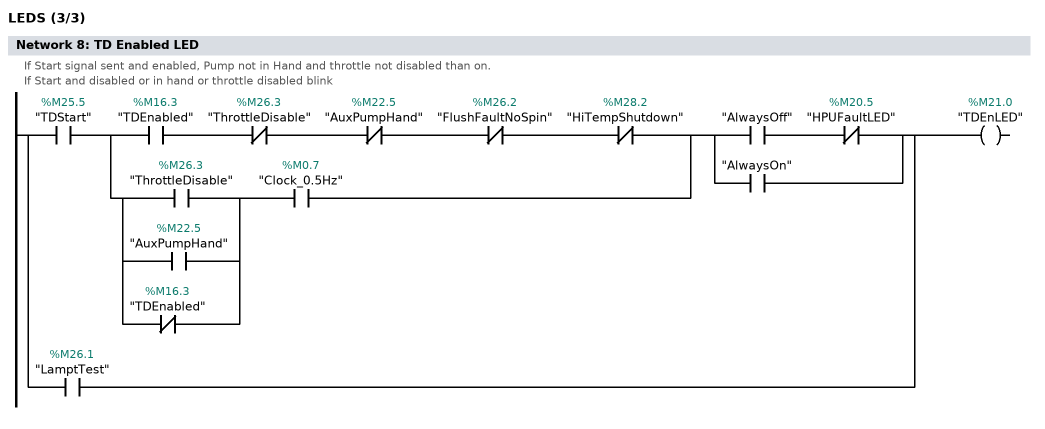
   RUNG wire#powerrail
      Contact( "TDStart" )
      wire#w1
      Contact( "TDEnabled" )
      I_Contact( "ThrottleDisable" )
      I_Contact( "AuxPumpHand" )
      I_Contact( "FlushFaultNoSpin" )
      I_Contact( "HiTempShutdown" )
      wire#w2
      Contact( "AlwaysOff" )
      I_Contact( "HPUFaultLED" )
      wire#w4
      Coil( "TDEnLED" )
   END_RUNG
   RUNG wire#w1
      Contact( "ThrottleDisable" )
      wire#w3
      Contact( "Clock_0.5Hz" )
   END_RUNG wire#w2
   RUNG wire#w1
      Contact( "AuxPumpHand" )
   END_RUNG wire#w3
   RUNG wire#w1
      I_Contact( "TDEnabled" )
   END_RUNG wire#w3
   RUNG wire#w2
      Contact( "AlwaysOn" )
   END_RUNG wire#w4
   RUNG wire#powerrail
      Contact( "LamptTest" )
   END_RUNG wire#w4
   // the same network as SCL:
   "TDEnLED" := ("TDStart" AND (("TDEnabled" AND NOT "ThrottleDisable" AND NOT "AuxPumpHand" AND NOT "FlushFaultNoSpin" AND NOT "HiTempShutdown") OR (("ThrottleDisable" OR "AuxPumpHand" OR NOT "TDEnabled") AND "Clock_0.5Hz")) AND (("AlwaysOff" AND NOT "HPUFaultLED") OR "AlwaysOn")) OR "LamptTest";
END_REGION
END_FUNCTION_BLOCK

FUNCTION_BLOCK "Timers"   // FB21, LAD
TITLE = Timers
{ S7_Optimized_Access := 'TRUE' }
// Written By Kristopher Gimenez March 3rd,2023
// 
// This block and its DB will contain the system runtimes logic and data
// stored: AutoNumber false, MemoryReserve 100, SetENOAutomatically false
   VAR
      TDTimeReset : Bool;   // Bit set from HMI used to reset time
      M1TimeReset : Bool;   // Bit set from HMI used to reset time
      M2TimeReset : Bool;   // Bit set from HMI used to reset time
      AuxTimeReset : Bool;   // Bit set from HMI used to reset time
      CoolerTimeReset : Bool;   // Bit set from HMI used to reset time
      TDRuntime : "Runtime_Out";
      M1Runtime { S7_SetPoint := 'True'} : "Runtime_Out";
      M2Runtime { S7_SetPoint := 'True'} : "Runtime_Out";
      AuxRuntime { S7_SetPoint := 'True'} : "Runtime_Out";
      CoolerRuntime { S7_SetPoint := 'True'} : "Runtime_Out";
      SystemRunStart : Bool;
      System_Runtime { S7_SetPoint := 'True'} : "Runtime";
      M1_Runtime { S7_SetPoint := 'True'} : "Runtime";
      M2_Runtime { S7_SetPoint := 'True'} : "Runtime";
      Cooler_Runtime { S7_SetPoint := 'True'} : "Runtime";
      AuxPump_Runtime { S7_SetPoint := 'True'} : "Runtime";
   END_VAR
BEGIN

REGION Network 1: TD Run Time
   // Call Each cycle. Reset from HMI
